   DATA[2646,2] := 2.0;
   DATA[2646,3] := 2.0;
   DATA[2646,4] := 262.3366;
   DATA[2646,5] := 8.393873;
   DATA[2646,6] := 329.2745;
   DATA[2646,7] := 2.455131;
   DATA[2646,8] := 2.0;
   DATA[2646,9] := 2.0;
   DATA[2646,10] := 2.0;
   DATA[2646,11] := 19.69396;
   DATA[2646,12] := 2.209397;
   DATA[2646,13] := 833.5603;
   DATA[2646,14] := 1.0;
   DATA[2646,15] := 2.0;
   DATA[2646,16] := 1.0;
   DATA[2646,17] := 1.0;
   DATA[2646,18] := 1.0;
   DATA[2646,19] := 2.0;
   DATA[2646,20] := 148.808;
   DATA[2646,21] := 155.191;
   DATA[2646,22] := 1.717105;
   DATA[2646,23] := 880.3127;
   DATA[2646,24] := 2.0;
   DATA[2646,25] := 2.0;
   DATA[2646,26] := 7.873815;
   DATA[2646,27] := 144.7578;
   DATA[2646,28] := 261.3753;
   DATA[2646,29] := 12.07383;
   DATA[2646,30] := 1.725711;
   DATA[2646,31] := 1.28705;
   DATA[2646,32] := 0.7352687;
   DATA[2646,33] := 0.3066329;
   DATA[2646,34] := 2.0;
   DATA[2646,35] := 250.2403;
   DATA[2646,36] := 1.665972;
   DATA[2646,37] := 189.022;
   DATA[2646,38] := 0.000128152;
   DATA[2646,39] := 1.0;
   DATA[2646,40] := 1.0;
   DATA[2647,0] := 2.595202;
   DATA[2647,1] := 869.8411;
   DATA[2647,2] := 2.0;
   DATA[2647,3] := 2.0;
   DATA[2647,4] := 262.3366;
   DATA[2647,5] := 8.393873;
   DATA[2647,6] := 329.2745;
   DATA[2647,7] := 2.454362;
   DATA[2647,8] := 2.0;
   DATA[2647,9] := 2.0;
   DATA[2647,10] := 2.0;
   DATA[2647,11] := 19.69396;
   DATA[2647,12] := 2.209397;
   DATA[2647,13] := 833.4402;
   DATA[2647,14] := 1.0;
   DATA[2647,15] := 2.0;
   DATA[2647,16] := 1.0;
   DATA[2647,17] := 1.0;
   DATA[2647,18] := 1.0;
   DATA[2647,19] := 2.0;
   DATA[2647,20] := 148.808;
   DATA[2647,21] := 155.191;
   DATA[2647,22] := 1.718002;
   DATA[2647,23] := 880.8895;
   DATA[2647,24] := 2.0;
   DATA[2647,25] := 2.0;
   DATA[2647,26] := 7.873815;
   DATA[2647,27] := 144.7578;
   DATA[2647,28] := 261.3753;
   DATA[2647,29] := 12.03538;
   DATA[2647,30] := 1.726096;
   DATA[2647,31] := 1.281286;
   DATA[2647,32] := 0.7352687;
   DATA[2647,33] := 0.3065048;
   DATA[2647,34] := 2.0;
   DATA[2647,35] := 250.2403;
   DATA[2647,36] := 1.730048;
   DATA[2647,37] := 189.1182;
   DATA[2647,38] := 0.000128152;
   DATA[2647,39] := 1.0;
   DATA[2647,40] := 1.0;
   DATA[2648,0] := 2.620504;
   DATA[2648,1] := 869.4094;
   DATA[2648,2] := 2.0;
   DATA[2648,3] := 2.0;
   DATA[2648,4] := 262.3366;
   DATA[2648,5] := 8.393873;
   DATA[2648,6] := 329.2745;
   DATA[2648,7] := 2.45308;
   DATA[2648,8] := 2.0;
   DATA[2648,9] := 2.0;
   DATA[2648,10] := 2.0;
   DATA[2648,11] := 19.66835;
   DATA[2648,12] := 2.209397;
   DATA[2648,13] := 833.6404;
   DATA[2648,14] := 1.0;
   DATA[2648,15] := 2.0;
   DATA[2648,16] := 1.0;
   DATA[2648,17] := 1.0;
   DATA[2648,18] := 1.0;
   DATA[2648,19] := 2.0;
   DATA[2648,20] := 148.808;
   DATA[2648,21] := 155.191;
   DATA[2648,22] := 1.718387;
   DATA[2648,23] := 880.8895;
   DATA[2648,24] := 2.0;
   DATA[2648,25] := 2.0;
   DATA[2648,26] := 7.873815;
   DATA[2648,27] := 144.7578;
   DATA[2648,28] := 261.183;
   DATA[2648,29] := 12.03538;
   DATA[2648,30] := 1.726993;
   DATA[2648,31] := 1.28103;
   DATA[2648,32] := 0.7352687;
   DATA[2648,33] := 0.3065048;
   DATA[2648,34] := 2.0;
   DATA[2648,35] := 250.2403;
   DATA[2648,36] := 1.730048;
   DATA[2648,37] := 189.1182;
   DATA[2648,38] := 0.000128152;
   DATA[2648,39] := 1.0;
   DATA[2648,40] := 1.0;
   DATA[2649,0] := 2.656055;
   DATA[2649,1] := 869.4879;
   DATA[2649,2] := 2.0;
   DATA[2649,3] := 2.0;
   DATA[2649,4] := 262.3366;
   DATA[2649,5] := 8.393873;
   DATA[2649,6] := 329.2745;
   DATA[2649,7] := 2.45308;
   DATA[2649,8] := 2.0;
   DATA[2649,9] := 2.0;
   DATA[2649,10] := 2.0;
   DATA[2649,11] := 19.66835;
   DATA[2649,12] := 2.209397;
   DATA[2649,13] := 833.36;
   DATA[2649,14] := 1.0;
   DATA[2649,15] := 2.0;
   DATA[2649,16] := 1.0;
   DATA[2649,17] := 1.0;
   DATA[2649,18] := 1.0;
   DATA[2649,19] := 2.0;
   DATA[2649,20] := 148.808;
   DATA[2649,21] := 155.191;
   DATA[2649,22] := 1.720437;
   DATA[2649,23] := 881.1587;
   DATA[2649,24] := 2.0;
   DATA[2649,25] := 2.0;
   DATA[2649,26] := 7.874776;
   DATA[2649,27] := 144.7578;
   DATA[2649,28] := 261.183;
   DATA[2649,29] := 12.03538;
   DATA[2649,30] := 1.726993;
   DATA[2649,31] := 1.28103;
   DATA[2649,32] := 0.7352687;
   DATA[2649,33] := 0.3065048;
   DATA[2649,34] := 2.0;
   DATA[2649,35] := 250.2403;
   DATA[2649,36] := 1.730048;
   DATA[2649,37] := 189.1182;
   DATA[2649,38] := 0.000128152;
   DATA[2649,39] := 1.0;
   DATA[2649,40] := 1.0;
   DATA[2650,0] := 2.665663;
   DATA[2650,1] := 869.4094;
   DATA[2650,2] := 2.0;
   DATA[2650,3] := 2.0;
   DATA[2650,4] := 262.3366;
   DATA[2650,5] := 8.396757;
   DATA[2650,6] := 329.2745;
   DATA[2650,7] := 2.45308;
   DATA[2650,8] := 2.0;
   DATA[2650,9] := 2.0;
   DATA[2650,10] := 2.0;
   DATA[2650,11] := 19.74198;
   DATA[2650,12] := 2.209397;
   DATA[2650,13] := 833.36;
   DATA[2650,14] := 1.0;
   DATA[2650,15] := 2.0;
   DATA[2650,16] := 1.0;
   DATA[2650,17] := 1.0;
   DATA[2650,18] := 1.0;
   DATA[2650,19] := 2.0;
   DATA[2650,20] := 148.808;
   DATA[2650,21] := 155.191;
   DATA[2650,22] := 1.720437;
   DATA[2650,23] := 881.0433;
   DATA[2650,24] := 2.0;
   DATA[2650,25] := 2.0;
   DATA[2650,26] := 7.874776;
   DATA[2650,27] := 144.7578;
   DATA[2650,28] := 261.183;
   DATA[2650,29] := 12.03538;
   DATA[2650,30] := 1.727634;
   DATA[2650,31] := 1.273601;
   DATA[2650,32] := 0.7352687;
   DATA[2650,33] := 0.3065048;
   DATA[2650,34] := 2.0;
   DATA[2650,35] := 250.3525;
   DATA[2650,36] := 1.730048;
   DATA[2650,37] := 189.1182;
   DATA[2650,38] := 0.000128152;
   DATA[2650,39] := 1.0;
   DATA[2650,40] := 1.0;
   DATA[2651,0] := 2.665663;
   DATA[2651,1] := 869.5271;
   DATA[2651,2] := 2.0;
   DATA[2651,3] := 2.0;
   DATA[2651,4] := 262.3366;
   DATA[2651,5] := 8.396757;
   DATA[2651,6] := 329.1464;
   DATA[2651,7] := 2.454618;
   DATA[2651,8] := 2.0;
   DATA[2651,9] := 2.0;
   DATA[2651,10] := 2.0;
   DATA[2651,11] := 19.74198;
   DATA[2651,12] := 2.209397;
   DATA[2651,13] := 833.5603;
   DATA[2651,14] := 1.0;
   DATA[2651,15] := 2.0;
   DATA[2651,16] := 1.0;
   DATA[2651,17] := 1.0;
   DATA[2651,18] := 1.0;
   DATA[2651,19] := 2.0;
   DATA[2651,20] := 148.808;
   DATA[2651,21] := 155.191;
   DATA[2651,22] := 1.720437;
   DATA[2651,23] := 881.0433;
   DATA[2651,24] := 2.0;
   DATA[2651,25] := 2.0;
   DATA[2651,26] := 7.874776;
   DATA[2651,27] := 144.7578;
   DATA[2651,28] := 261.183;
   DATA[2651,29] := 12.03538;
   DATA[2651,30] := 1.728916;
   DATA[2651,31] := 1.277699;
   DATA[2651,32] := 0.7352687;
   DATA[2651,33] := 0.3065048;
   DATA[2651,34] := 2.0;
   DATA[2651,35] := 250.3525;
   DATA[2651,36] := 1.730048;
   DATA[2651,37] := 189.1182;
   DATA[2651,38] := 0.000128152;
   DATA[2651,39] := 1.0;
   DATA[2651,40] := 1.0;
   DATA[2652,0] := 2.65061;
   DATA[2652,1] := 869.8019;
   DATA[2652,2] := 2.0;
   DATA[2652,3] := 2.0;
   DATA[2652,4] := 262.3366;
   DATA[2652,5] := 8.396757;
   DATA[2652,6] := 329.1464;
   DATA[2652,7] := 2.454618;
   DATA[2652,8] := 2.0;
   DATA[2652,9] := 2.0;
   DATA[2652,10] := 2.0;
   DATA[2652,11] := 19.74198;
   DATA[2652,12] := 2.209397;
   DATA[2652,13] := 833.6004;
   DATA[2652,14] := 1.0;
   DATA[2652,15] := 2.0;
   DATA[2652,16] := 1.0;
   DATA[2652,17] := 1.0;
   DATA[2652,18] := 1.0;
   DATA[2652,19] := 2.0;
   DATA[2652,20] := 148.808;
   DATA[2652,21] := 155.191;
   DATA[2652,22] := 1.720437;
   DATA[2652,23] := 881.1202;
   DATA[2652,24] := 2.0;
   DATA[2652,25] := 2.0;
   DATA[2652,26] := 7.874776;
   DATA[2652,27] := 144.6039;
   DATA[2652,28] := 261.2151;
   DATA[2652,29] := 12.03538;
   DATA[2652,30] := 1.7293;
   DATA[2652,31] := 1.293711;
   DATA[2652,32] := 0.7352687;
   DATA[2652,33] := 0.3065048;
   DATA[2652,34] := 2.0;
   DATA[2652,35] := 250.3525;
   DATA[2652,36] := 1.730048;
   DATA[2652,37] := 189.1182;
   DATA[2652,38] := 0.000128152;
   DATA[2652,39] := 1.0;
   DATA[2652,40] := 1.0;
   DATA[2653,0] := 2.62755;
   DATA[2653,1] := 869.8019;
   DATA[2653,2] := 2.0;
   DATA[2653,3] := 2.0;
   DATA[2653,4] := 262.3366;
   DATA[2653,5] := 8.396757;
   DATA[2653,6] := 329.1464;
   DATA[2653,7] := 2.455515;
   DATA[2653,8] := 2.0;
   DATA[2653,9] := 2.0;
   DATA[2653,10] := 2.0;
   DATA[2653,11] := 19.67476;
   DATA[2653,12] := 2.209397;
   DATA[2653,13] := 833.4802;
   DATA[2653,14] := 1.0;
   DATA[2653,15] := 2.0;
   DATA[2653,16] := 1.0;
   DATA[2653,17] := 1.0;
   DATA[2653,18] := 1.0;
   DATA[2653,19] := 2.0;
   DATA[2653,20] := 148.808;
   DATA[2653,21] := 155.191;
   DATA[2653,22] := 1.720437;
   DATA[2653,23] := 880.8895;
   DATA[2653,24] := 2.0;
   DATA[2653,25] := 2.0;
   DATA[2653,26] := 7.874776;
   DATA[2653,27] := 144.6039;
   DATA[2653,28] := 261.3432;
   DATA[2653,29] := 12.03538;
   DATA[2653,30] := 1.7293;
   DATA[2653,31] := 1.297041;
   DATA[2653,32] := 0.7352687;
   DATA[2653,33] := 0.3065048;
   DATA[2653,34] := 2.0;
   DATA[2653,35] := 250.3525;
   DATA[2653,36] := 1.730048;
   DATA[2653,37] := 189.1182;
   DATA[2653,38] := 0.000128152;
   DATA[2653,39] := 1.0;
   DATA[2653,40] := 1.0;
   DATA[2654,0] := 2.622746;
   DATA[2654,1] := 869.8411;
   DATA[2654,2] := 2.0;
   DATA[2654,3] := 2.0;
   DATA[2654,4] := 262.3366;
   DATA[2654,5] := 8.396757;
   DATA[2654,6] := 329.1464;
   DATA[2654,7] := 2.455515;
   DATA[2654,8] := 2.0;
   DATA[2654,9] := 2.0;
   DATA[2654,10] := 2.0;
   DATA[2654,11] := 19.67476;
   DATA[2654,12] := 2.209397;
   DATA[2654,13] := 833.7606;
   DATA[2654,14] := 1.0;
   DATA[2654,15] := 2.0;
   DATA[2654,16] := 1.0;
   DATA[2654,17] := 1.0;
   DATA[2654,18] := 1.0;
   DATA[2654,19] := 2.0;
   DATA[2654,20] := 148.808;
   DATA[2654,21] := 155.191;
   DATA[2654,22] := 1.720437;
   DATA[2654,23] := 880.7357;
   DATA[2654,24] := 2.0;
   DATA[2654,25] := 2.0;
   DATA[2654,26] := 7.874776;
   DATA[2654,27] := 144.6039;
   DATA[2654,28] := 261.3432;
   DATA[2654,29] := 12.03538;
   DATA[2654,30] := 1.7293;
   DATA[2654,31] := 1.296401;
   DATA[2654,32] := 0.7352687;
   DATA[2654,33] := 0.3065689;
   DATA[2654,34] := 2.0;
   DATA[2654,35] := 250.3525;
   DATA[2654,36] := 1.730048;
   DATA[2654,37] := 189.1342;
   DATA[2654,38] := 0.000128152;
   DATA[2654,39] := 1.0;
   DATA[2654,40] := 1.0;
   DATA[2655,0] := 2.607693;
   DATA[2655,1] := 869.4094;
   DATA[2655,2] := 2.0;
   DATA[2655,3] := 2.0;
   DATA[2655,4] := 262.3366;
   DATA[2655,5] := 8.396757;
   DATA[2655,6] := 329.1464;
   DATA[2655,7] := 2.455515;
   DATA[2655,8] := 2.0;
   DATA[2655,9] := 2.0;
   DATA[2655,10] := 2.0;
   DATA[2655,11] := 19.62033;
   DATA[2655,12] := 2.209397;
   DATA[2655,13] := 833.6404;
   DATA[2655,14] := 1.0;
   DATA[2655,15] := 2.0;
   DATA[2655,16] := 1.0;
   DATA[2655,17] := 1.0;
   DATA[2655,18] := 1.0;
   DATA[2655,19] := 2.0;
   DATA[2655,20] := 148.808;
   DATA[2655,21] := 155.3961;
   DATA[2655,22] := 1.720437;
   DATA[2655,23] := 880.928;
   DATA[2655,24] := 2.0;
   DATA[2655,25] := 2.0;
   DATA[2655,26] := 7.874776;
   DATA[2655,27] := 144.6039;
   DATA[2655,28] := 261.3432;
   DATA[2655,29] := 12.03538;
   DATA[2655,30] := 1.7293;
   DATA[2655,31] := 1.296016;
   DATA[2655,32] := 0.7352687;
   DATA[2655,33] := 0.3066329;
   DATA[2655,34] := 2.0;
   DATA[2655,35] := 250.3525;
   DATA[2655,36] := 1.730048;
   DATA[2655,37] := 189.1662;
   DATA[2655,38] := 0.000128152;
   DATA[2655,39] := 1.0;
   DATA[2655,40] := 1.0;
   DATA[2656,0] := 2.587516;
   DATA[2656,1] := 869.8411;
   DATA[2656,2] := 2.0;
   DATA[2656,3] := 2.0;
   DATA[2656,4] := 262.3366;
   DATA[2656,5] := 8.396757;
   DATA[2656,6] := 329.1464;
   DATA[2656,7] := 2.455515;
   DATA[2656,8] := 2.0;
   DATA[2656,9] := 2.0;
   DATA[2656,10] := 2.0;
   DATA[2656,11] := 19.62033;
   DATA[2656,12] := 2.208884;
   DATA[2656,13] := 833.5603;
   DATA[2656,14] := 1.0;
   DATA[2656,15] := 2.0;
   DATA[2656,16] := 1.0;
   DATA[2656,17] := 1.0;
   DATA[2656,18] := 1.0;
   DATA[2656,19] := 2.0;
   DATA[2656,20] := 148.808;
   DATA[2656,21] := 155.3961;
   DATA[2656,22] := 1.720437;
   DATA[2656,23] := 880.7357;
   DATA[2656,24] := 2.0;
   DATA[2656,25] := 2.0;
   DATA[2656,26] := 7.874776;
   DATA[2656,27] := 144.6039;
   DATA[2656,28] := 261.3432;
   DATA[2656,29] := 12.03538;
   DATA[2656,30] := 1.7293;
   DATA[2656,31] := 1.292558;
   DATA[2656,32] := 0.7352687;
   DATA[2656,33] := 0.3066329;
   DATA[2656,34] := 2.0;
   DATA[2656,35] := 250.3525;
   DATA[2656,36] := 1.730048;
   DATA[2656,37] := 189.1662;
   DATA[2656,38] := 0.000128152;
   DATA[2656,39] := 1.0;
   DATA[2656,40] := 1.0;
   DATA[2657,0] := 2.562854;
   DATA[2657,1] := 870.0767;
   DATA[2657,2] := 2.0;
   DATA[2657,3] := 2.0;
   DATA[2657,4] := 262.3366;
   DATA[2657,5] := 8.396757;
   DATA[2657,6] := 329.1464;
   DATA[2657,7] := 2.455515;
   DATA[2657,8] := 2.0;
   DATA[2657,9] := 2.0;
   DATA[2657,10] := 2.0;
   DATA[2657,11] := 19.57232;
   DATA[2657,12] := 2.208884;
   DATA[2657,13] := 834.0009;
   DATA[2657,14] := 1.0;
   DATA[2657,15] := 2.0;
   DATA[2657,16] := 1.0;
   DATA[2657,17] := 1.0;
   DATA[2657,18] := 1.0;
   DATA[2657,19] := 2.0;
   DATA[2657,20] := 148.808;
   DATA[2657,21] := 155.3961;
   DATA[2657,22] := 1.720437;
   DATA[2657,23] := 880.4666;
   DATA[2657,24] := 2.0;
   DATA[2657,25] := 2.0;
   DATA[2657,26] := 7.873815;
   DATA[2657,27] := 144.6039;
   DATA[2657,28] := 261.3432;
   DATA[2657,29] := 12.03538;
   DATA[2657,30] := 1.7293;
   DATA[2657,31] := 1.291533;
   DATA[2657,32] := 0.7352687;
   DATA[2657,33] := 0.3066329;
   DATA[2657,34] := 2.0;
   DATA[2657,35] := 250.1762;
   DATA[2657,36] := 1.730048;
   DATA[2657,37] := 189.1662;
   DATA[2657,38] := 0.000128152;
   DATA[2657,39] := 1.0;
   DATA[2657,40] := 1.0;
   DATA[2658,0] := 2.537873;
   DATA[2658,1] := 869.7234;
   DATA[2658,2] := 2.0;
   DATA[2658,3] := 2.0;
   DATA[2658,4] := 262.3366;
   DATA[2658,5] := 8.396757;
   DATA[2658,6] := 329.1464;
   DATA[2658,7] := 2.452952;
   DATA[2658,8] := 2.0;
   DATA[2658,9] := 2.0;
   DATA[2658,10] := 2.0;
   DATA[2658,11] := 19.57232;
   DATA[2658,12] := 2.208884;
   DATA[2658,13] := 834.0009;
   DATA[2658,14] := 1.0;
   DATA[2658,15] := 2.0;
   DATA[2658,16] := 1.0;
   DATA[2658,17] := 1.0;
   DATA[2658,18] := 1.0;
   DATA[2658,19] := 2.0;
   DATA[2658,20] := 148.808;
   DATA[2658,21] := 155.3961;
   DATA[2658,22] := 1.720437;
   DATA[2658,23] := 880.8511;
   DATA[2658,24] := 2.0;
   DATA[2658,25] := 2.0;
   DATA[2658,26] := 7.873815;
   DATA[2658,27] := 144.6039;
   DATA[2658,28] := 261.3432;
   DATA[2658,29] := 12.03538;
   DATA[2658,30] := 1.7293;
   DATA[2658,31] := 1.291533;
   DATA[2658,32] := 0.7352687;
   DATA[2658,33] := 0.3066329;
   DATA[2658,34] := 2.0;
   DATA[2658,35] := 250.1762;
   DATA[2658,36] := 1.730048;
   DATA[2658,37] := 188.9419;
   DATA[2658,38] := 0.000128152;
   DATA[2658,39] := 1.0;
   DATA[2658,40] := 1.0;
   DATA[2659,0] := 2.521218;
   DATA[2659,1] := 869.8019;
   DATA[2659,2] := 2.0;
   DATA[2659,3] := 2.0;
   DATA[2659,4] := 262.3366;
   DATA[2659,5] := 8.396757;
   DATA[2659,6] := 329.1464;
   DATA[2659,7] := 2.452952;
   DATA[2659,8] := 2.0;
   DATA[2659,9] := 2.0;
   DATA[2659,10] := 2.0;
   DATA[2659,11] := 19.62674;
   DATA[2659,12] := 2.209653;
   DATA[2659,13] := 834.0009;
   DATA[2659,14] := 1.0;
   DATA[2659,15] := 2.0;
   DATA[2659,16] := 1.0;
   DATA[2659,17] := 1.0;
   DATA[2659,18] := 1.0;
   DATA[2659,19] := 2.0;
   DATA[2659,20] := 148.808;
   DATA[2659,21] := 155.3961;
   DATA[2659,22] := 1.718002;
   DATA[2659,23] := 880.6588;
   DATA[2659,24] := 2.0;
   DATA[2659,25] := 2.0;
   DATA[2659,26] := 7.872853;
   DATA[2659,27] := 144.6039;
   DATA[2659,28] := 261.3432;
   DATA[2659,29] := 12.03538;
   DATA[2659,30] := 1.7293;
   DATA[2659,31] := 1.291533;
   DATA[2659,32] := 0.7352687;
   DATA[2659,33] := 0.3066329;
   DATA[2659,34] := 2.0;
   DATA[2659,35] := 249.9519;
   DATA[2659,36] := 1.730048;
   DATA[2659,37] := 188.8618;
   DATA[2659,38] := 0.000128152;
   DATA[2659,39] := 1.0;
   DATA[2659,40] := 1.0;
   DATA[2660,0] := 2.500721;
   DATA[2660,1] := 869.9196;
   DATA[2660,2] := 2.0;
   DATA[2660,3] := 2.0;
   DATA[2660,4] := 262.3366;
   DATA[2660,5] := 8.396757;
   DATA[2660,6] := 329.1464;
   DATA[2660,7] := 2.452952;
   DATA[2660,8] := 2.0;
   DATA[2660,9] := 2.0;
   DATA[2660,10] := 2.0;
   DATA[2660,11] := 19.62674;
   DATA[2660,12] := 2.209653;
   DATA[2660,13] := 834.1611;
   DATA[2660,14] := 1.0;
   DATA[2660,15] := 2.0;
   DATA[2660,16] := 1.0;
   DATA[2660,17] := 1.0;
   DATA[2660,18] := 1.0;
   DATA[2660,19] := 2.0;
   DATA[2660,20] := 148.808;
   DATA[2660,21] := 155.3961;
   DATA[2660,22] := 1.717361;
   DATA[2660,23] := 881.0818;
   DATA[2660,24] := 2.0;
   DATA[2660,25] := 2.0;
   DATA[2660,26] := 7.872853;
   DATA[2660,27] := 144.6039;
   DATA[2660,28] := 261.3432;
   DATA[2660,29] := 12.03538;
   DATA[2660,30] := 1.7293;
   DATA[2660,31] := 1.28436;
   DATA[2660,32] := 0.7352687;
   DATA[2660,33] := 0.3066329;
   DATA[2660,34] := 2.0;
   DATA[2660,35] := 249.9519;
   DATA[2660,36] := 1.730048;
   DATA[2660,37] := 188.8618;
   DATA[2660,38] := 0.000128152;
   DATA[2660,39] := 1.0;
   DATA[2660,40] := 1.0;
   DATA[2661,0] := 2.483426;
   DATA[2661,1] := 870.1159;
   DATA[2661,2] := 2.0;
   DATA[2661,3] := 2.0;
   DATA[2661,4] := 262.3366;
   DATA[2661,5] := 8.396757;
   DATA[2661,6] := 329.1464;
   DATA[2661,7] := 2.452952;
   DATA[2661,8] := 2.0;
   DATA[2661,9] := 2.0;
   DATA[2661,10] := 2.0;
   DATA[2661,11] := 19.62674;
   DATA[2661,12] := 2.209653;
   DATA[2661,13] := 833.6004;
   DATA[2661,14] := 1.0;
   DATA[2661,15] := 2.0;
   DATA[2661,16] := 1.0;
   DATA[2661,17] := 1.0;
   DATA[2661,18] := 1.0;
   DATA[2661,19] := 2.0;
   DATA[2661,20] := 148.808;
   DATA[2661,21] := 155.3961;
   DATA[2661,22] := 1.717233;
   DATA[2661,23] := 880.7742;
   DATA[2661,24] := 2.0;
   DATA[2661,25] := 2.0;
   DATA[2661,26] := 7.872853;
   DATA[2661,27] := 144.7065;
   DATA[2661,28] := 261.3432;
   DATA[2661,29] := 12.03538;
   DATA[2661,30] := 1.7293;
   DATA[2661,31] := 1.286922;
   DATA[2661,32] := 0.7352687;
   DATA[2661,33] := 0.3066329;
   DATA[2661,34] := 2.0;
   DATA[2661,35] := 249.9519;
   DATA[2661,36] := 1.730048;
   DATA[2661,37] := 188.8618;
   DATA[2661,38] := 0.000128152;
   DATA[2661,39] := 1.0;
   DATA[2661,40] := 1.0;
   DATA[2662,0] := 2.468052;
   DATA[2662,1] := 870.2729;
   DATA[2662,2] := 2.0;
   DATA[2662,3] := 2.0;
   DATA[2662,4] := 262.3366;
   DATA[2662,5] := 8.396757;
   DATA[2662,6] := 329.1464;
   DATA[2662,7] := 2.452952;
   DATA[2662,8] := 2.0;
   DATA[2662,9] := 2.0;
   DATA[2662,10] := 2.0;
   DATA[2662,11] := 19.67476;
   DATA[2662,12] := 2.208756;
   DATA[2662,13] := 833.5603;
   DATA[2662,14] := 1.0;
   DATA[2662,15] := 2.0;
   DATA[2662,16] := 1.0;
   DATA[2662,17] := 1.0;
   DATA[2662,18] := 1.0;
   DATA[2662,19] := 2.0;
   DATA[2662,20] := 148.808;
   DATA[2662,21] := 155.3961;
   DATA[2662,22] := 1.717233;
   DATA[2662,23] := 880.5819;
   DATA[2662,24] := 2.0;
   DATA[2662,25] := 2.0;
   DATA[2662,26] := 7.872853;
   DATA[2662,27] := 144.7065;
   DATA[2662,28] := 261.3432;
   DATA[2662,29] := 12.03538;
   DATA[2662,30] := 1.7293;
   DATA[2662,31] := 1.301012;
   DATA[2662,32] := 0.7352687;
   DATA[2662,33] := 0.3066329;
   DATA[2662,34] := 2.0;
   DATA[2662,35] := 249.9519;
   DATA[2662,36] := 1.730048;
   DATA[2662,37] := 188.8618;
   DATA[2662,38] := 0.000128152;
   DATA[2662,39] := 1.0;
   DATA[2662,40] := 1.0;
   DATA[2663,0] := 2.449156;
   DATA[2663,1] := 870.5084;
   DATA[2663,2] := 2.0;
   DATA[2663,3] := 2.0;
   DATA[2663,4] := 262.3366;
   DATA[2663,5] := 8.396757;
   DATA[2663,6] := 329.1464;
   DATA[2663,7] := 2.452952;
   DATA[2663,8] := 2.0;
   DATA[2663,9] := 2.0;
   DATA[2663,10] := 2.0;
   DATA[2663,11] := 19.69396;
   DATA[2663,12] := 2.208756;
   DATA[2663,13] := 833.8007;
   DATA[2663,14] := 1.0;
   DATA[2663,15] := 2.0;
   DATA[2663,16] := 1.0;
   DATA[2663,17] := 1.0;
   DATA[2663,18] := 1.0;
   DATA[2663,19] := 2.0;
   DATA[2663,20] := 148.808;
   DATA[2663,21] := 155.3961;
   DATA[2663,22] := 1.717233;
   DATA[2663,23] := 880.6973;
   DATA[2663,24] := 2.0;
   DATA[2663,25] := 2.0;
   DATA[2663,26] := 7.872853;
   DATA[2663,27] := 144.7065;
   DATA[2663,28] := 261.3432;
   DATA[2663,29] := 12.03538;
   DATA[2663,30] := 1.7293;
   DATA[2663,31] := 1.296529;
   DATA[2663,32] := 0.7352687;
   DATA[2663,33] := 0.3066329;
   DATA[2663,34] := 2.0;
   DATA[2663,35] := 249.9519;
   DATA[2663,36] := 1.730048;
   DATA[2663,37] := 188.8618;
   DATA[2663,38] := 0.000128152;
   DATA[2663,39] := 1.0;
   DATA[2663,40] := 1.0;
   DATA[2664,0] := 2.436665;
   DATA[2664,1] := 870.4299;
   DATA[2664,2] := 2.0;
   DATA[2664,3] := 2.0;
   DATA[2664,4] := 262.3366;
   DATA[2664,5] := 8.396757;
   DATA[2664,6] := 329.1464;
   DATA[2664,7] := 2.452055;
   DATA[2664,8] := 2.0;
   DATA[2664,9] := 2.0;
   DATA[2664,10] := 2.0;
   DATA[2664,11] := 19.69396;
   DATA[2664,12] := 2.206322;
   DATA[2664,13] := 834.0009;
   DATA[2664,14] := 1.0;
   DATA[2664,15] := 2.0;
   DATA[2664,16] := 1.0;
   DATA[2664,17] := 1.0;
   DATA[2664,18] := 1.0;
   DATA[2664,19] := 2.0;
   DATA[2664,20] := 148.808;
   DATA[2664,21] := 155.3961;
   DATA[2664,22] := 1.717233;
   DATA[2664,23] := 880.7357;
   DATA[2664,24] := 2.0;
   DATA[2664,25] := 2.0;
   DATA[2664,26] := 7.872853;
   DATA[2664,27] := 144.7065;
   DATA[2664,28] := 261.3432;
   DATA[2664,29] := 12.03538;
   DATA[2664,30] := 1.726352;
   DATA[2664,31] := 1.3005;
   DATA[2664,32] := 0.7352687;
   DATA[2664,33] := 0.3066329;
   DATA[2664,34] := 2.0;
   DATA[2664,35] := 250.016;
   DATA[2664,36] := 1.730048;
   DATA[2664,37] := 188.8618;
   DATA[2664,38] := 0.000128152;
   DATA[2664,39] := 1.0;
   DATA[2664,40] := 1.0;
   DATA[2665,0] := 2.431861;
   DATA[2665,1] := 870.5869;
   DATA[2665,2] := 2.0;
   DATA[2665,3] := 2.0;
   DATA[2665,4] := 262.3366;
   DATA[2665,5] := 8.396757;
   DATA[2665,6] := 329.1464;
   DATA[2665,7] := 2.451799;
   DATA[2665,8] := 2.0;
   DATA[2665,9] := 2.0;
   DATA[2665,10] := 2.0;
   DATA[2665,11] := 19.69396;
   DATA[2665,12] := 2.206322;
   DATA[2665,13] := 834.4415;
   DATA[2665,14] := 1.0;
   DATA[2665,15] := 2.0;
   DATA[2665,16] := 1.0;
   DATA[2665,17] := 1.0;
   DATA[2665,18] := 1.0;
   DATA[2665,19] := 2.0;
   DATA[2665,20] := 148.808;
   DATA[2665,21] := 155.3961;
   DATA[2665,22] := 1.717233;
   DATA[2665,23] := 881.2356;
   DATA[2665,24] := 2.0;
   DATA[2665,25] := 2.0;
   DATA[2665,26] := 7.872853;
   DATA[2665,27] := 144.7065;
   DATA[2665,28] := 261.3432;
   DATA[2665,29] := 12.03538;
   DATA[2665,30] := 1.726352;
   DATA[2665,31] := 1.3119;
   DATA[2665,32] := 0.7352687;
   DATA[2665,33] := 0.3066329;
   DATA[2665,34] := 2.0;
   DATA[2665,35] := 250.0961;
   DATA[2665,36] := 1.730048;
   DATA[2665,37] := 188.8618;
   DATA[2665,38] := 0.000128152;
   DATA[2665,39] := 1.0;
   DATA[2665,40] := 1.0;
   DATA[2666,0] := 2.431861;
   DATA[2666,1] := 870.4692;
   DATA[2666,2] := 2.0;
   DATA[2666,3] := 2.0;
   DATA[2666,4] := 262.3366;
   DATA[2666,5] := 8.396757;
   DATA[2666,6] := 329.1464;
   DATA[2666,7] := 2.451799;
   DATA[2666,8] := 2.0;
   DATA[2666,9] := 2.0;
   DATA[2666,10] := 2.0;
   DATA[2666,11] := 19.72598;
   DATA[2666,12] := 2.206322;
   DATA[2666,13] := 834.4415;
   DATA[2666,14] := 1.0;
   DATA[2666,15] := 2.0;
   DATA[2666,16] := 1.0;
   DATA[2666,17] := 1.0;
   DATA[2666,18] := 1.0;
   DATA[2666,19] := 2.0;
   DATA[2666,20] := 148.808;
   DATA[2666,21] := 155.3961;
   DATA[2666,22] := 1.717233;
   DATA[2666,23] := 881.4663;
   DATA[2666,24] := 2.0;
   DATA[2666,25] := 2.0;
   DATA[2666,26] := 7.872853;
   DATA[2666,27] := 144.7065;
   DATA[2666,28] := 261.3432;
   DATA[2666,29] := 12.03538;
   DATA[2666,30] := 1.726352;
   DATA[2666,31] := 1.30652;
   DATA[2666,32] := 0.7352687;
   DATA[2666,33] := 0.3066329;
   DATA[2666,34] := 2.0;
   DATA[2666,35] := 250.0961;
   DATA[2666,36] := 1.730048;
   DATA[2666,37] := 188.8618;
   DATA[2666,38] := 0.000128152;
   DATA[2666,39] := 1.0;
   DATA[2666,40] := 1.0;
   DATA[2667,0] := 2.455882;
   DATA[2667,1] := 870.5869;
   DATA[2667,2] := 2.0;
   DATA[2667,3] := 2.0;
   DATA[2667,4] := 262.3366;
   DATA[2667,5] := 8.396757;
   DATA[2667,6] := 329.1464;
   DATA[2667,7] := 2.455131;
   DATA[2667,8] := 2.0;
   DATA[2667,9] := 2.0;
   DATA[2667,10] := 2.0;
   DATA[2667,11] := 19.74198;
   DATA[2667,12] := 2.20645;
   DATA[2667,13] := 834.802;
   DATA[2667,14] := 1.0;
   DATA[2667,15] := 2.0;
   DATA[2667,16] := 1.0;
   DATA[2667,17] := 1.0;
   DATA[2667,18] := 1.0;
   DATA[2667,19] := 2.0;
   DATA[2667,20] := 148.808;
   DATA[2667,21] := 155.3961;
   DATA[2667,22] := 1.719156;
   DATA[2667,23] := 882.0431;
   DATA[2667,24] := 2.0;
   DATA[2667,25] := 2.0;
   DATA[2667,26] := 7.872853;
   DATA[2667,27] := 144.7065;
   DATA[2667,28] := 261.3432;
   DATA[2667,29] := 12.03538;
   DATA[2667,30] := 1.726352;
   DATA[2667,31] := 1.311387;
   DATA[2667,32] := 0.7352687;
   DATA[2667,33] := 0.3066329;
   DATA[2667,34] := 2.0;
   DATA[2667,35] := 250.1442;
   DATA[2667,36] := 1.730048;
   DATA[2667,37] := 188.8618;
   DATA[2667,38] := 0.000128152;
   DATA[2667,39] := 1.0;
   DATA[2667,40] := 1.0;
   DATA[2668,0] := 2.50008;
   DATA[2668,1] := 870.3907;
   DATA[2668,2] := 2.0;
   DATA[2668,3] := 2.0;
   DATA[2668,4] := 262.3366;
   DATA[2668,5] := 8.396757;
   DATA[2668,6] := 329.1464;
   DATA[2668,7] := 2.455131;
   DATA[2668,8] := 2.0;
   DATA[2668,9] := 2.0;
   DATA[2668,10] := 2.0;
   DATA[2668,11] := 19.75799;
   DATA[2668,12] := 2.209909;
   DATA[2668,13] := 834.802;
   DATA[2668,14] := 1.0;
   DATA[2668,15] := 2.0;
   DATA[2668,16] := 1.0;
   DATA[2668,17] := 1.0;
   DATA[2668,18] := 1.0;
   DATA[2668,19] := 2.0;
   DATA[2668,20] := 148.808;
   DATA[2668,21] := 155.3961;
   DATA[2668,22] := 1.719156;
   DATA[2668,23] := 882.1969;
   DATA[2668,24] := 2.0;
   DATA[2668,25] := 2.0;
   DATA[2668,26] := 7.872853;
   DATA[2668,27] := 144.7065;
   DATA[2668,28] := 261.3432;
   DATA[2668,29] := 12.03538;
   DATA[2668,30] := 1.726352;
   DATA[2668,31] := 1.313949;
   DATA[2668,32] := 0.7352687;
   DATA[2668,33] := 0.3066329;
   DATA[2668,34] := 2.0;
   DATA[2668,35] := 250.3044;
   DATA[2668,36] := 1.730048;
   DATA[2668,37] := 189.0381;
   DATA[2668,38] := 0.000128152;
   DATA[2668,39] := 1.0;
   DATA[2668,40] := 1.0;
   DATA[2669,0] := 2.537873;
   DATA[2669,1] := 870.7047;
   DATA[2669,2] := 2.0;
   DATA[2669,3] := 2.0;
   DATA[2669,4] := 262.3366;
   DATA[2669,5] := 8.396757;
   DATA[2669,6] := 329.1464;
   DATA[2669,7] := 2.455131;
   DATA[2669,8] := 2.0;
   DATA[2669,9] := 2.0;
   DATA[2669,10] := 2.0;
   DATA[2669,11] := 19.7964;
   DATA[2669,12] := 2.209909;
   DATA[2669,13] := 835.1625;
   DATA[2669,14] := 1.0;
   DATA[2669,15] := 2.0;
   DATA[2669,16] := 1.0;
   DATA[2669,17] := 1.0;
   DATA[2669,18] := 1.0;
   DATA[2669,19] := 2.0;
   DATA[2669,20] := 148.808;
   DATA[2669,21] := 155.3961;
   DATA[2669,22] := 1.719156;
   DATA[2669,23] := 882.2354;
   DATA[2669,24] := 2.0;
   DATA[2669,25] := 2.0;
   DATA[2669,26] := 7.874135;
   DATA[2669,27] := 144.7065;
   DATA[2669,28] := 261.3432;
   DATA[2669,29] := 12.03538;
   DATA[2669,30] := 1.726352;
   DATA[2669,31] := 1.311643;
   DATA[2669,32] := 0.7352687;
   DATA[2669,33] := 0.3066329;
   DATA[2669,34] := 2.0;
   DATA[2669,35] := 250.3044;
   DATA[2669,36] := 1.730048;
   DATA[2669,37] := 189.0541;
   DATA[2669,38] := 0.000128152;
   DATA[2669,39] := 1.0;
   DATA[2669,40] := 1.0;
   DATA[2670,0] := 2.585594;
   DATA[2670,1] := 871.058;
   DATA[2670,2] := 2.0;
   DATA[2670,3] := 2.0;
   DATA[2670,4] := 262.3366;
   DATA[2670,5] := 8.396757;
   DATA[2670,6] := 329.1464;
   DATA[2670,7] := 2.455131;
   DATA[2670,8] := 2.0;
   DATA[2670,9] := 2.0;
   DATA[2670,10] := 2.0;
   DATA[2670,11] := 19.7964;
   DATA[2670,12] := 2.209909;
   DATA[2670,13] := 835.1625;
   DATA[2670,14] := 1.0;
   DATA[2670,15] := 2.0;
   DATA[2670,16] := 1.0;
   DATA[2670,17] := 1.0;
   DATA[2670,18] := 1.0;
   DATA[2670,19] := 2.0;
   DATA[2670,20] := 148.808;
   DATA[2670,21] := 155.3961;
   DATA[2670,22] := 1.717105;
   DATA[2670,23] := 882.3892;
   DATA[2670,24] := 2.0;
   DATA[2670,25] := 2.0;
   DATA[2670,26] := 7.874135;
   DATA[2670,27] := 144.7065;
   DATA[2670,28] := 261.3432;
   DATA[2670,29] := 12.03538;
   DATA[2670,30] := 1.726352;
   DATA[2670,31] := 1.288587;
   DATA[2670,32] := 0.7352687;
   DATA[2670,33] := 0.3066329;
   DATA[2670,34] := 2.0;
   DATA[2670,35] := 250.3044;
   DATA[2670,36] := 1.730048;
   DATA[2670,37] := 189.1182;
   DATA[2670,38] := 0.000128152;
   DATA[2670,39] := 1.0;
   DATA[2670,40] := 1.0;
   DATA[2671,0] := 2.618903;
   DATA[2671,1] := 870.7047;
   DATA[2671,2] := 2.0;
   DATA[2671,3] := 2.0;
   DATA[2671,4] := 262.3366;
   DATA[2671,5] := 8.396757;
   DATA[2671,6] := 329.1464;
   DATA[2671,7] := 2.456156;
   DATA[2671,8] := 2.0;
   DATA[2671,9] := 2.0;
   DATA[2671,10] := 2.0;
   DATA[2671,11] := 19.7804;
   DATA[2671,12] := 2.209909;
   DATA[2671,13] := 835.2025;
   DATA[2671,14] := 1.0;
   DATA[2671,15] := 2.0;
   DATA[2671,16] := 1.0;
   DATA[2671,17] := 1.0;
   DATA[2671,18] := 1.0;
   DATA[2671,19] := 2.0;
   DATA[2671,20] := 148.808;
   DATA[2671,21] := 155.3961;
   DATA[2671,22] := 1.717105;
   DATA[2671,23] := 882.6967;
   DATA[2671,24] := 2.0;
   DATA[2671,25] := 2.0;
   DATA[2671,26] := 7.874135;
   DATA[2671,27] := 144.7065;
   DATA[2671,28] := 261.3432;
   DATA[2671,29] := 12.03538;
   DATA[2671,30] := 1.726352;
   DATA[2671,31] := 1.27296;
   DATA[2671,32] := 0.7352687;
   DATA[2671,33] := 0.3066329;
   DATA[2671,34] := 2.0;
   DATA[2671,35] := 250.3044;
   DATA[2671,36] := 1.730048;
   DATA[2671,37] := 189.1182;
   DATA[2671,38] := 0.000128152;
   DATA[2671,39] := 1.0;
   DATA[2671,40] := 1.0;
   DATA[2672,0] := 2.644845;
   DATA[2672,1] := 871.2542;
   DATA[2672,2] := 2.0;
   DATA[2672,3] := 2.0;
   DATA[2672,4] := 262.3366;
   DATA[2672,5] := 8.396757;
   DATA[2672,6] := 329.1464;
   DATA[2672,7] := 2.456156;
   DATA[2672,8] := 2.0;
   DATA[2672,9] := 2.0;
   DATA[2672,10] := 2.0;
   DATA[2672,11] := 19.73558;
   DATA[2672,12] := 2.209909;
   DATA[2672,13] := 835.2827;
   DATA[2672,14] := 1.0;
   DATA[2672,15] := 2.0;
   DATA[2672,16] := 1.0;
   DATA[2672,17] := 1.0;
   DATA[2672,18] := 1.0;
   DATA[2672,19] := 2.0;
   DATA[2672,20] := 148.808;
   DATA[2672,21] := 155.3961;
   DATA[2672,22] := 1.717105;
   DATA[2672,23] := 882.8121;
   DATA[2672,24] := 2.0;
   DATA[2672,25] := 2.0;
   DATA[2672,26] := 7.874135;
   DATA[2672,27] := 144.7065;
   DATA[2672,28] := 261.3432;
   DATA[2672,29] := 12.03538;
   DATA[2672,30] := 1.726352;
   DATA[2672,31] := 1.265915;
   DATA[2672,32] := 0.7352687;
   DATA[2672,33] := 0.3066329;
   DATA[2672,34] := 2.0;
   DATA[2672,35] := 250.3044;
   DATA[2672,36] := 1.730048;
   DATA[2672,37] := 188.9419;
   DATA[2672,38] := 0.000128152;
   DATA[2672,39] := 1.0;
   DATA[2672,40] := 1.0;
   DATA[2673,0] := 2.658937;
   DATA[2673,1] := 871.058;
   DATA[2673,3] := 2.0;
   DATA[2673,4] := 262.3366;
   DATA[2673,5] := 8.396757;
   DATA[2673,6] := 329.1464;
   DATA[2673,7] := 2.456156;
   DATA[2673,8] := 2.0;
   DATA[2673,9] := 2.0;
   DATA[2673,10] := 2.0;
   DATA[2673,11] := 19.71637;
   DATA[2673,12] := 2.211959;
   DATA[2673,13] := 835.6832;
   DATA[2673,14] := 1.0;
   DATA[2673,15] := 2.0;
   DATA[2673,16] := 1.0;
   DATA[2673,17] := 1.0;
   DATA[2673,18] := 1.0;
   DATA[2673,19] := 2.0;
   DATA[2673,20] := 148.808;
   DATA[2673,21] := 155.3961;
   DATA[2673,22] := 1.717105;
   DATA[2673,23] := 882.6967;
   DATA[2673,24] := 2.0;
   DATA[2673,25] := 2.0;
   DATA[2673,26] := 7.874135;
   DATA[2673,27] := 144.7065;
   DATA[2673,28] := 261.3432;
   DATA[2673,29] := 12.03538;
   DATA[2673,30] := 1.728659;
   DATA[2673,31] := 1.261944;
   DATA[2673,32] := 0.7352687;
   DATA[2673,33] := 0.3066329;
   DATA[2673,34] := 2.0;
   DATA[2673,35] := 250.3044;
   DATA[2673,36] := 1.730048;
   DATA[2673,37] := 188.9419;
   DATA[2673,38] := 0.000128152;
   DATA[2673,39] := 1.0;
   DATA[2673,40] := 1.0;
   DATA[2674,0] := 2.658937;
   DATA[2674,1] := 871.0972;
   DATA[2674,3] := 2.0;
   DATA[2674,4] := 262.3366;
   DATA[2674,5] := 8.396757;
   DATA[2674,6] := 329.1464;
   DATA[2674,7] := 2.453978;
   DATA[2674,8] := 2.0;
   DATA[2674,9] := 2.0;
   DATA[2674,10] := 2.0;
   DATA[2674,11] := 19.71637;
   DATA[2674,12] := 2.212215;
   DATA[2674,13] := 835.563;
   DATA[2674,14] := 1.0;
   DATA[2674,15] := 2.0;
   DATA[2674,16] := 1.0;
   DATA[2674,17] := 1.0;
   DATA[2674,18] := 1.0;
   DATA[2674,19] := 2.0;
   DATA[2674,20] := 148.808;
   DATA[2674,21] := 155.3961;
   DATA[2674,22] := 1.717105;
   DATA[2674,23] := 882.889;
   DATA[2674,24] := 2.0;
   DATA[2674,25] := 2.0;
   DATA[2674,26] := 7.874135;
   DATA[2674,27] := 144.7065;
   DATA[2674,28] := 261.3432;
   DATA[2674,29] := 12.03538;
   DATA[2674,30] := 1.728916;
   DATA[2674,31] := 1.276419;
   DATA[2674,32] := 0.7352687;
   DATA[2674,33] := 0.3066329;
   DATA[2674,34] := 2.0;
   DATA[2674,35] := 250.1442;
   DATA[2674,36] := 1.730048;
   DATA[2674,37] := 188.9419;
   DATA[2674,38] := 0.000128152;
   DATA[2674,39] := 1.0;
   DATA[2674,40] := 1.0;
   DATA[2675,0] := 2.639721;
   DATA[2675,1] := 871.215;
   DATA[2675,3] := 2.0;
   DATA[2675,4] := 262.3366;
   DATA[2675,5] := 8.396757;
   DATA[2675,6] := 329.1464;
   DATA[2675,7] := 2.452952;
   DATA[2675,8] := 2.0;
   DATA[2675,9] := 2.0;
   DATA[2675,10] := 2.0;
   DATA[2675,11] := 19.71637;
   DATA[2675,12] := 2.212215;
   DATA[2675,13] := 835.4028;
   DATA[2675,14] := 1.0;
   DATA[2675,15] := 2.0;
   DATA[2675,16] := 1.0;
   DATA[2675,17] := 1.0;
   DATA[2675,18] := 1.0;
   DATA[2675,19] := 2.0;
   DATA[2675,20] := 148.808;
   DATA[2675,21] := 155.3961;
   DATA[2675,22] := 1.717105;
   DATA[2675,23] := 882.6198;
   DATA[2675,24] := 2.0;
   DATA[2675,25] := 2.0;
   DATA[2675,26] := 7.874135;
   DATA[2675,27] := 144.7065;
   DATA[2675,28] := 261.3432;
   DATA[2675,29] := 11.72776;
   DATA[2675,30] := 1.728916;
   DATA[2675,31] := 1.28167;
   DATA[2675,32] := 0.7352687;
   DATA[2675,33] := 0.3066329;
   DATA[2675,34] := 2.0;
   DATA[2675,35] := 250.1442;
   DATA[2675,36] := 1.730048;
   DATA[2675,37] := 188.9419;
   DATA[2675,38] := 0.000128152;
   DATA[2675,39] := 1.0;
   DATA[2675,40] := 1.0;
   DATA[2676,0] := 2.633635;
   DATA[2676,1] := 870.9794;
   DATA[2676,3] := 2.0;
   DATA[2676,4] := 262.3366;
   DATA[2676,5] := 8.396757;
   DATA[2676,6] := 329.1464;
   DATA[2676,7] := 2.452952;
   DATA[2676,8] := 2.0;
   DATA[2676,9] := 2.0;
   DATA[2676,10] := 2.0;
   DATA[2676,11] := 19.71637;
   DATA[2676,12] := 2.209397;
   DATA[2676,13] := 835.6031;
   DATA[2676,14] := 1.0;
   DATA[2676,15] := 2.0;
   DATA[2676,16] := 1.0;
   DATA[2676,17] := 1.0;
   DATA[2676,18] := 1.0;
   DATA[2676,19] := 2.0;
   DATA[2676,20] := 148.808;
   DATA[2676,21] := 155.5242;
   DATA[2676,22] := 1.717105;
   DATA[2676,23] := 882.5814;
   DATA[2676,24] := 2.0;
   DATA[2676,25] := 2.0;
   DATA[2676,26] := 7.874135;
   DATA[2676,27] := 144.7065;
   DATA[2676,28] := 261.3432;
   DATA[2676,29] := 11.72776;
   DATA[2676,30] := 1.728916;
   DATA[2676,31] := 1.276547;
   DATA[2676,32] := 0.7352687;
   DATA[2676,33] := 0.3066329;
   DATA[2676,34] := 2.0;
   DATA[2676,35] := 250.3525;
   DATA[2676,36] := 1.730048;
   DATA[2676,37] := 189.1182;
   DATA[2676,38] := 0.000128152;
   DATA[2676,39] := 1.0;
   DATA[2676,40] := 1.0;
   DATA[2677,0] := 2.633635;
   DATA[2677,1] := 870.6654;
   DATA[2677,3] := 2.0;
   DATA[2677,4] := 262.3366;
   DATA[2677,5] := 8.396757;
   DATA[2677,6] := 329.1464;
   DATA[2677,7] := 2.452952;
   DATA[2677,8] := 2.0;
   DATA[2677,9] := 2.0;
   DATA[2677,10] := 2.0;
   DATA[2677,11] := 19.71637;
   DATA[2677,12] := 2.209397;
   DATA[2677,13] := 835.4429;
   DATA[2677,14] := 1.0;
   DATA[2677,15] := 2.0;
   DATA[2677,16] := 1.0;
   DATA[2677,17] := 1.0;
   DATA[2677,18] := 1.0;
   DATA[2677,19] := 2.0;
   DATA[2677,20] := 148.808;
   DATA[2677,21] := 155.5242;
   DATA[2677,22] := 1.718515;
   DATA[2677,23] := 882.6967;
   DATA[2677,24] := 2.0;
   DATA[2677,25] := 2.0;
   DATA[2677,26] := 7.874135;
   DATA[2677,27] := 144.7065;
   DATA[2677,28] := 261.3432;
   DATA[2677,29] := 11.72776;
   DATA[2677,30] := 1.730838;
   DATA[2677,31] := 1.280902;
   DATA[2677,32] := 0.7352687;
   DATA[2677,33] := 0.3084905;
   DATA[2677,34] := 2.0;
   DATA[2677,35] := 250.3525;
   DATA[2677,36] := 1.730048;
   DATA[2677,37] := 189.1182;
   DATA[2677,38] := 0.000128152;
   DATA[2677,39] := 1.0;
   DATA[2677,40] := 1.0;
   DATA[2678,0] := 2.625628;
   DATA[2678,1] := 870.6654;
   DATA[2678,3] := 2.0;
   DATA[2678,4] := 262.3366;
   DATA[2678,5] := 8.396757;
   DATA[2678,6] := 329.1464;
   DATA[2678,7] := 2.452952;
   DATA[2678,8] := 2.0;
   DATA[2678,9] := 2.0;
   DATA[2678,10] := 2.0;
   DATA[2678,11] := 19.73878;
   DATA[2678,12] := 2.209397;
   DATA[2678,13] := 835.3627;
   DATA[2678,14] := 1.0;
   DATA[2678,15] := 2.0;
   DATA[2678,16] := 1.0;
   DATA[2678,17] := 1.0;
   DATA[2678,18] := 1.0;
   DATA[2678,19] := 2.0;
   DATA[2678,20] := 148.808;
   DATA[2678,21] := 155.5242;
   DATA[2678,22] := 1.718515;
   DATA[2678,23] := 882.6583;
   DATA[2678,24] := 2.0;
   DATA[2678,25] := 2.0;
   DATA[2678,26] := 7.874135;
   DATA[2678,27] := 144.7065;
   DATA[2678,28] := 261.3432;
   DATA[2678,29] := 12.07383;
   DATA[2678,30] := 1.731735;
   DATA[2678,31] := 1.288203;
   DATA[2678,32] := 0.7352687;
   DATA[2678,33] := 0.3084905;
   DATA[2678,34] := 2.0;
   DATA[2678,35] := 250.4967;
   DATA[2678,36] := 1.730048;
   DATA[2678,37] := 189.2624;
   DATA[2678,38] := 0.000128152;
   DATA[2678,39] := 1.0;
   DATA[2678,40] := 1.0;
   DATA[2679,0] := 2.600006;
   DATA[2679,1] := 871.058;
   DATA[2679,3] := 2.0;
   DATA[2679,4] := 262.3366;
   DATA[2679,5] := 8.396757;
   DATA[2679,6] := 329.1464;
   DATA[2679,7] := 2.452952;
   DATA[2679,8] := 2.0;
   DATA[2679,9] := 2.0;
   DATA[2679,10] := 2.0;
   DATA[2679,11] := 19.74838;
   DATA[2679,12] := 2.209397;
   DATA[2679,13] := 835.0023;
   DATA[2679,14] := 1.0;
   DATA[2679,15] := 2.0;
   DATA[2679,16] := 1.0;
   DATA[2679,17] := 1.0;
   DATA[2679,18] := 1.0;
   DATA[2679,19] := 2.0;
   DATA[2679,20] := 148.808;
   DATA[2679,21] := 155.473;
   DATA[2679,22] := 1.718515;
   DATA[2679,23] := 882.4661;
   DATA[2679,24] := 2.0;
   DATA[2679,25] := 2.0;
   DATA[2679,26] := 7.874135;
   DATA[2679,27] := 144.7065;
   DATA[2679,28] := 261.3432;
   DATA[2679,29] := 12.07383;
   DATA[2679,30] := 1.731735;
   DATA[2679,31] := 1.307416;
   DATA[2679,32] := 0.7352687;
   DATA[2679,33] := 0.3084905;
   DATA[2679,34] := 2.0;
   DATA[2679,35] := 250.4967;
   DATA[2679,36] := 1.730048;
   DATA[2679,37] := 189.2624;
   DATA[2679,38] := 0.000128152;
   DATA[2679,39] := 1.0;
   DATA[2679,40] := 1.0;
   DATA[2680,0] := 2.552285;
   DATA[2680,1] := 870.7047;
   DATA[2680,3] := 2.0;
   DATA[2680,4] := 262.3366;
   DATA[2680,5] := 8.396757;
   DATA[2680,6] := 329.0182;
   DATA[2680,7] := 2.452568;
   DATA[2680,8] := 2.0;
   DATA[2680,9] := 2.0;
   DATA[2680,10] := 2.0;
   DATA[2680,11] := 19.74838;
   DATA[2680,12] := 2.20645;
   DATA[2680,13] := 834.762;
   DATA[2680,14] := 1.0;
   DATA[2680,15] := 2.0;
   DATA[2680,16] := 1.0;
   DATA[2680,17] := 1.0;
   DATA[2680,18] := 1.0;
   DATA[2680,19] := 2.0;
   DATA[2680,20] := 148.808;
   DATA[2680,21] := 155.4473;
   DATA[2680,22] := 1.718515;
   DATA[2680,23] := 882.5045;
   DATA[2680,24] := 2.0;
   DATA[2680,25] := 2.0;
   DATA[2680,26] := 7.870931;
   DATA[2680,27] := 144.7834;
   DATA[2680,28] := 261.3432;
   DATA[2680,29] := 12.07383;
   DATA[2680,30] := 1.731735;
   DATA[2680,31] := 1.320994;
   DATA[2680,32] := 0.7352687;
   DATA[2680,33] := 0.3084905;
   DATA[2680,34] := 2.0;
   DATA[2680,35] := 250.4967;
   DATA[2680,36] := 1.730048;
   DATA[2680,37] := 189.2624;
   DATA[2680,38] := 0.000128152;
   DATA[2680,39] := 1.0;
   DATA[2680,40] := 1.0;
   DATA[2681,0] := 2.499119;
   DATA[2681,1] := 870.8224;
   DATA[2681,3] := 2.0;
   DATA[2681,4] := 262.3366;
   DATA[2681,5] := 8.396757;
   DATA[2681,6] := 329.0182;
   DATA[2681,7] := 2.451671;
   DATA[2681,8] := 2.0;
   DATA[2681,9] := 2.0;
   DATA[2681,10] := 2.0;
   DATA[2681,11] := 19.74838;
   DATA[2681,12] := 2.20645;
   DATA[2681,13] := 834.6818;
   DATA[2681,14] := 1.0;
   DATA[2681,15] := 2.0;
   DATA[2681,16] := 1.0;
   DATA[2681,17] := 1.0;
   DATA[2681,18] := 1.0;
   DATA[2681,19] := 2.0;
   DATA[2681,20] := 148.808;
   DATA[2681,21] := 155.4473;
   DATA[2681,22] := 1.718515;
   DATA[2681,23] := 882.12;
   DATA[2681,24] := 2.0;
   DATA[2681,25] := 2.0;
   DATA[2681,26] := 7.870931;
   DATA[2681,27] := 144.7834;
   DATA[2681,28] := 261.3432;
   DATA[2681,29] := 12.07383;
   DATA[2681,30] := 1.731735;
   DATA[2681,31] := 1.329064;
   DATA[2681,32] := 0.7352687;
   DATA[2681,33] := 0.3084905;
   DATA[2681,34] := 2.0;
   DATA[2681,35] := 250.4967;
   DATA[2681,36] := 1.730048;
   DATA[2681,37] := 189.2624;
   DATA[2681,38] := 0.000128152;
   DATA[2681,39] := 1.0;
   DATA[2681,40] := 1.0;
   DATA[2682,0] := 2.400154;
   DATA[2682,1] := 870.6654;
   DATA[2682,2] := 1.0;
   DATA[2682,3] := 2.0;
   DATA[2682,4] := 262.3366;
   DATA[2682,5] := 8.396757;
   DATA[2682,6] := 329.0182;
   DATA[2682,7] := 2.451671;
   DATA[2682,8] := 2.0;
   DATA[2682,9] := 2.0;
   DATA[2682,10] := 2.0;
   DATA[2682,11] := 19.74838;
   DATA[2682,12] := 2.20645;
   DATA[2682,13] := 835.2025;
   DATA[2682,14] := 1.0;
   DATA[2682,15] := 2.0;
   DATA[2682,16] := 1.0;
   DATA[2682,17] := 1.0;
   DATA[2682,18] := 1.0;
   DATA[2682,19] := 2.0;
   DATA[2682,20] := 148.808;
   DATA[2682,21] := 155.4473;
   DATA[2682,22] := 1.718515;
   DATA[2682,23] := 882.2738;
   DATA[2682,24] := 2.0;
   DATA[2682,25] := 2.0;
   DATA[2682,26] := 7.873815;
   DATA[2682,27] := 144.7834;
   DATA[2682,28] := 261.3432;
   DATA[2682,29] := 12.07383;
   DATA[2682,30] := 1.731351;
   DATA[2682,31] := 1.332138;
   DATA[2682,32] := 0.7352687;
   DATA[2682,33] := 0.3084905;
   DATA[2682,34] := 2.0;
   DATA[2682,35] := 250.4967;
   DATA[2682,36] := 1.730048;
   DATA[2682,37] := 189.2624;
   DATA[2682,38] := 0.000128152;
   DATA[2682,39] := 1.0;
   DATA[2682,40] := 1.0;
   DATA[2683,0] := 2.223361;
   DATA[2683,1] := 870.9794;
   DATA[2683,2] := 1.0;
   DATA[2683,3] := 2.0;
   DATA[2683,4] := 262.3366;
   DATA[2683,5] := 8.396757;
   DATA[2683,6] := 329.0182;
   DATA[2683,7] := 2.451671;
   DATA[2683,8] := 2.0;
   DATA[2683,9] := 2.0;
   DATA[2683,10] := 2.0;
   DATA[2683,11] := 19.74838;
   DATA[2683,12] := 2.20645;
   DATA[2683,13] := 834.6818;
   DATA[2683,14] := 1.0;
   DATA[2683,15] := 2.0;
   DATA[2683,16] := 1.0;
   DATA[2683,17] := 1.0;
   DATA[2683,18] := 1.0;
   DATA[2683,19] := 2.0;
   DATA[2683,20] := 148.808;
   DATA[2683,21] := 155.4473;
   DATA[2683,22] := 1.718515;
   DATA[2683,23] := 882.5045;
   DATA[2683,24] := 2.0;
   DATA[2683,25] := 2.0;
   DATA[2683,26] := 7.874776;
   DATA[2683,27] := 144.7834;
   DATA[2683,28] := 261.3432;
   DATA[2683,29] := 12.07383;
   DATA[2683,30] := 1.731351;
   DATA[2683,31] := 1.31523;
   DATA[2683,32] := 0.7352687;
   DATA[2683,33] := 0.3084905;
   DATA[2683,34] := 2.0;
   DATA[2683,35] := 250.4967;
   DATA[2683,36] := 1.810143;
   DATA[2683,37] := 189.2624;
   DATA[2683,38] := 0.000128152;
   DATA[2683,39] := 1.0;
   DATA[2683,40] := 1.0;
   DATA[2684,0] := 1.916216;
   DATA[2684,1] := 870.5869;
   DATA[2684,2] := 1.0;
   DATA[2684,3] := 2.0;
   DATA[2684,4] := 262.3366;
   DATA[2684,5] := 8.396757;
   DATA[2684,6] := 329.0182;
   DATA[2684,7] := 2.451671;
   DATA[2684,8] := 2.0;
   DATA[2684,9] := 2.0;
   DATA[2684,10] := 2.0;
   DATA[2684,11] := 19.74838;
   DATA[2684,12] := 2.207091;
   DATA[2684,13] := 835.2025;
   DATA[2684,14] := 1.0;
   DATA[2684,15] := 2.0;
   DATA[2684,16] := 1.0;
   DATA[2684,17] := 1.0;
   DATA[2684,18] := 1.0;
   DATA[2684,19] := 2.0;
   DATA[2684,20] := 148.808;
   DATA[2684,21] := 155.3961;
   DATA[2684,22] := 1.716592;
   DATA[2684,23] := 882.5045;
   DATA[2684,24] := 2.0;
   DATA[2684,25] := 2.0;
   DATA[2684,26] := 7.874776;
   DATA[2684,27] := 144.7834;
   DATA[2684,28] := 261.3432;
   DATA[2684,29] := 12.07383;
   DATA[2684,30] := 1.729557;
   DATA[2684,31] := 1.311387;
   DATA[2684,32] := 0.7352687;
   DATA[2684,33] := 0.3084905;
   DATA[2684,34] := 2.0;
   DATA[2684,35] := 250.4967;
   DATA[2684,36] := 1.810143;
   DATA[2684,37] := 189.2624;
   DATA[2684,38] := 0.000128152;
   DATA[2684,39] := 1.0;
   DATA[2684,40] := 1.0;
   DATA[2685,0] := 1.582808;
   DATA[2685,1] := 870.8224;
   DATA[2685,2] := 1.0;
   DATA[2685,3] := 2.0;
   DATA[2685,4] := 262.3366;
   DATA[2685,5] := 8.396757;
   DATA[2685,6] := 329.0182;
   DATA[2685,7] := 2.452952;
   DATA[2685,8] := 2.0;
   DATA[2685,9] := 2.0;
   DATA[2685,10] := 2.0;
   DATA[2685,11] := 19.74838;
   DATA[2685,12] := 2.208756;
   DATA[2685,13] := 834.842;
   DATA[2685,14] := 1.0;
   DATA[2685,15] := 2.0;
   DATA[2685,16] := 1.0;
   DATA[2685,17] := 1.0;
   DATA[2685,18] := 1.0;
   DATA[2685,19] := 2.0;
   DATA[2685,20] := 148.808;
   DATA[2685,21] := 155.3961;
   DATA[2685,22] := 1.716592;
   DATA[2685,23] := 882.2738;
   DATA[2685,24] := 2.0;
   DATA[2685,25] := 2.0;
   DATA[2685,26] := 7.874776;
   DATA[2685,27] := 144.7834;
   DATA[2685,28] := 261.3432;
   DATA[2685,29] := 12.07383;
   DATA[2685,30] := 1.729557;
   DATA[2685,31] := 1.302677;
   DATA[2685,32] := 0.7352687;
   DATA[2685,33] := 0.3066329;
   DATA[2685,34] := 2.0;
   DATA[2685,35] := 250.4967;
   DATA[2685,36] := 1.810143;
   DATA[2685,37] := 189.2624;
   DATA[2685,38] := 0.000128152;
   DATA[2685,39] := 1.0;
   DATA[2685,40] := 1.0;
   DATA[2686,0] := 1.178618;
   DATA[2686,1] := 870.4299;
   DATA[2686,2] := 1.0;
   DATA[2686,3] := 2.0;
   DATA[2686,4] := 262.3366;
   DATA[2686,5] := 8.396757;
   DATA[2686,6] := 329.0182;
   DATA[2686,7] := 2.452952;
   DATA[2686,8] := 2.0;
   DATA[2686,9] := 2.0;
   DATA[2686,10] := 2.0;
   DATA[2686,11] := 19.69076;
   DATA[2686,12] := 2.209525;
   DATA[2686,13] := 835.1625;
   DATA[2686,14] := 1.0;
   DATA[2686,15] := 2.0;
   DATA[2686,16] := 1.0;
   DATA[2686,17] := 1.0;
   DATA[2686,18] := 1.0;
   DATA[2686,19] := 2.0;
   DATA[2686,20] := 148.808;
   DATA[2686,21] := 155.3961;
   DATA[2686,22] := 1.716592;
   DATA[2686,23] := 882.2738;
   DATA[2686,24] := 2.0;
   DATA[2686,25] := 2.0;
   DATA[2686,26] := 7.874776;
   DATA[2686,27] := 144.7834;
   DATA[2686,28] := 261.3432;
   DATA[2686,29] := 11.84312;
   DATA[2686,30] := 1.729557;
   DATA[2686,31] := 1.292814;
   DATA[2686,32] := 0.7352687;
   DATA[2686,33] := 0.3081703;
   DATA[2686,34] := 2.0;
   DATA[2686,35] := 250.4967;
   DATA[2686,36] := 1.730048;
   DATA[2686,37] := 189.2624;
   DATA[2686,38] := 0.000128152;
   DATA[2686,39] := 1.0;
   DATA[2686,40] := 1.0;
   DATA[2687,0] := 0.801012;
   DATA[2687,1] := 870.1944;
   DATA[2687,2] := 1.0;
   DATA[2687,3] := 2.0;
   DATA[2687,4] := 262.3366;
   DATA[2687,5] := 8.396757;
   DATA[2687,6] := 329.0182;
   DATA[2687,7] := 2.452952;
   DATA[2687,8] := 2.0;
   DATA[2687,9] := 2.0;
   DATA[2687,10] := 2.0;
   DATA[2687,11] := 19.69076;
   DATA[2687,12] := 2.209653;
   DATA[2687,13] := 835.0423;
   DATA[2687,14] := 1.0;
   DATA[2687,15] := 2.0;
   DATA[2687,16] := 1.0;
   DATA[2687,17] := 1.0;
   DATA[2687,18] := 1.0;
   DATA[2687,19] := 2.0;
   DATA[2687,20] := 148.808;
   DATA[2687,21] := 155.3961;
   DATA[2687,22] := 1.716592;
   DATA[2687,23] := 882.5814;
   DATA[2687,24] := 2.0;
   DATA[2687,25] := 2.0;
   DATA[2687,26] := 7.874776;
   DATA[2687,27] := 144.7834;
   DATA[2687,28] := 261.3432;
   DATA[2687,29] := 11.84312;
   DATA[2687,30] := 1.729557;
   DATA[2687,31] := 1.27834;
   DATA[2687,32] := 0.7352687;
   DATA[2687,33] := 0.3086827;
   DATA[2687,34] := 2.0;
   DATA[2687,35] := 250.4967;
   DATA[2687,36] := 1.730048;
   DATA[2687,37] := 189.2624;
   DATA[2687,38] := 0.000128152;
   DATA[2687,39] := 1.0;
   DATA[2687,40] := 1.0;
   DATA[2688,0] := 0.4829773;
   DATA[2688,1] := 869.8411;
   DATA[2688,2] := 1.0;
   DATA[2688,3] := 2.0;
   DATA[2688,4] := 262.3366;
   DATA[2688,5] := 8.396757;
   DATA[2688,6] := 329.0182;
   DATA[2688,7] := 2.452952;
   DATA[2688,8] := 2.0;
   DATA[2688,9] := 2.0;
   DATA[2688,10] := 2.0;
   DATA[2688,11] := 19.69076;
   DATA[2688,12] := 2.209653;
   DATA[2688,13] := 835.0423;
   DATA[2688,14] := 1.0;
   DATA[2688,15] := 2.0;
   DATA[2688,16] := 1.0;
   DATA[2688,17] := 1.0;
   DATA[2688,18] := 1.0;
   DATA[2688,19] := 2.0;
   DATA[2688,20] := 148.808;
   DATA[2688,21] := 155.3961;
   DATA[2688,22] := 1.716464;
   DATA[2688,23] := 882.8505;
   DATA[2688,24] := 2.0;
   DATA[2688,25] := 2.0;
   DATA[2688,26] := 7.874776;
   DATA[2688,27] := 144.7834;
   DATA[2688,28] := 261.3432;
   DATA[2688,29] := 11.84312;
   DATA[2688,30] := 1.729557;
   DATA[2688,31] := 1.257589;
   DATA[2688,32] := 0.7352687;
   DATA[2688,33] := 0.3086827;
   DATA[2688,34] := 2.0;
   DATA[2688,35] := 250.4967;
   DATA[2688,36] := 1.730048;
   DATA[2688,37] := 189.2624;
   DATA[2688,38] := 0.000128152;
   DATA[2688,39] := 1.0;
   DATA[2688,40] := 1.0;
   DATA[2689,0] := 0.2844057;
   DATA[2689,1] := 869.8804;
   DATA[2689,2] := 1.0;
   DATA[2689,3] := 2.0;
   DATA[2689,4] := 262.3366;
   DATA[2689,5] := 8.396757;
   DATA[2689,6] := 329.0182;
   DATA[2689,7] := 2.452952;
   DATA[2689,8] := 2.0;
   DATA[2689,9] := 2.0;
   DATA[2689,10] := 2.0;
   DATA[2689,11] := 19.69076;
   DATA[2689,12] := 2.209653;
   DATA[2689,13] := 835.2426;
   DATA[2689,14] := 1.0;
   DATA[2689,15] := 2.0;
   DATA[2689,16] := 1.0;
   DATA[2689,17] := 1.0;
   DATA[2689,18] := 1.0;
   DATA[2689,19] := 2.0;
   DATA[2689,20] := 148.808;
   DATA[2689,21] := 155.3961;
   DATA[2689,22] := 1.716464;
   DATA[2689,23] := 882.7736;
   DATA[2689,24] := 2.0;
   DATA[2689,25] := 2.0;
   DATA[2689,26] := 7.874776;
   DATA[2689,27] := 144.7834;
   DATA[2689,28] := 261.3432;
   DATA[2689,29] := 12.07383;
   DATA[2689,30] := 1.729557;
   DATA[2689,31] := 1.245805;
   DATA[2689,32] := 0.7352687;
   DATA[2689,33] := 0.3086827;
   DATA[2689,34] := 2.0;
   DATA[2689,35] := 250.3525;
   DATA[2689,36] := 1.730048;
   DATA[2689,37] := 189.1342;
   DATA[2689,38] := 0.000128152;
   DATA[2689,39] := 1.0;
   DATA[2689,40] := 1.0;
   DATA[2690,0] := 0.1518112;
   DATA[2690,1] := 869.8019;
   DATA[2690,2] := 1.0;
   DATA[2690,3] := 2.0;
   DATA[2690,4] := 262.3366;
   DATA[2690,5] := 8.396757;
   DATA[2690,6] := 329.0182;
   DATA[2690,7] := 2.452952;
   DATA[2690,8] := 2.0;
   DATA[2690,9] := 2.0;
   DATA[2690,10] := 2.0;
   DATA[2690,11] := 19.70677;
   DATA[2690,12] := 2.209653;
   DATA[2690,13] := 835.2025;
   DATA[2690,14] := 1.0;
   DATA[2690,15] := 2.0;
   DATA[2690,16] := 1.0;
   DATA[2690,17] := 1.0;
   DATA[2690,18] := 1.0;
   DATA[2690,19] := 2.0;
   DATA[2690,20] := 148.808;
   DATA[2690,21] := 155.3961;
   DATA[2690,22] := 1.716464;
   DATA[2690,23] := 882.7736;
   DATA[2690,24] := 2.0;
   DATA[2690,25] := 2.0;
   DATA[2690,26] := 7.874776;
   DATA[2690,27] := 144.7834;
   DATA[2690,28] := 261.3432;
   DATA[2690,29] := 12.22763;
   DATA[2690,30] := 1.731479;
   DATA[2690,31] := 1.244652;
   DATA[2690,32] := 0.7352687;
   DATA[2690,33] := 0.3086827;
   DATA[2690,34] := 2.0;
   DATA[2690,35] := 250.3525;
   DATA[2690,36] := 1.730048;
   DATA[2690,37] := 189.1342;
   DATA[2690,38] := 0.000128152;
   DATA[2690,39] := 1.0;
   DATA[2690,40] := 1.0;
   DATA[2691,0] := 0.07334337;
   DATA[2691,1] := 869.8411;
   DATA[2691,2] := 1.0;
   DATA[2691,3] := 2.0;
   DATA[2691,4] := 262.3366;
   DATA[2691,5] := 8.396757;
   DATA[2691,6] := 329.1207;
   DATA[2691,7] := 2.452952;
   DATA[2691,8] := 2.0;
   DATA[2691,9] := 2.0;
   DATA[2691,10] := 2.0;
   DATA[2691,11] := 19.74198;
   DATA[2691,12] := 2.209653;
   DATA[2691,13] := 835.4429;
   DATA[2691,14] := 1.0;
   DATA[2691,15] := 2.0;
   DATA[2691,16] := 1.0;
   DATA[2691,17] := 1.0;
   DATA[2691,18] := 1.0;
   DATA[2691,19] := 2.0;
   DATA[2691,20] := 148.808;
   DATA[2691,21] := 155.3961;
   DATA[2691,22] := 1.718515;
   DATA[2691,23] := 882.5045;
   DATA[2691,24] := 2.0;
   DATA[2691,25] := 2.0;
   DATA[2691,26] := 7.874776;
   DATA[2691,27] := 144.7834;
   DATA[2691,28] := 261.3432;
   DATA[2691,29] := 12.22763;
   DATA[2691,30] := 1.731479;
   DATA[2691,31] := 1.262713;
   DATA[2691,32] := 0.7352687;
   DATA[2691,33] := 0.3074016;
   DATA[2691,34] := 2.0;
   DATA[2691,35] := 250.2724;
   DATA[2691,36] := 1.730048;
   DATA[2691,37] := 188.958;
   DATA[2691,38] := 0.000128152;
   DATA[2691,39] := 1.0;
   DATA[2691,40] := 1.0;
   DATA[2692,0] := 0.02370048;
   DATA[2692,1] := 869.7234;
   DATA[2692,2] := 1.0;
   DATA[2692,3] := 2.0;
   DATA[2692,4] := 262.3366;
   DATA[2692,5] := 8.396757;
   DATA[2692,6] := 329.1207;
   DATA[2692,7] := 2.452952;
   DATA[2692,8] := 2.0;
   DATA[2692,9] := 2.0;
   DATA[2692,10] := 2.0;
   DATA[2692,11] := 19.74198;
   DATA[2692,12] := 2.209653;
   DATA[2692,13] := 835.4028;
   DATA[2692,14] := 1.0;
   DATA[2692,15] := 2.0;
   DATA[2692,16] := 1.0;
   DATA[2692,17] := 1.0;
   DATA[2692,18] := 1.0;
   DATA[2692,19] := 2.0;
   DATA[2692,20] := 148.808;
   DATA[2692,21] := 155.3961;
   DATA[2692,22] := 1.718515;
   DATA[2692,23] := 882.2738;
   DATA[2692,24] := 2.0;
   DATA[2692,25] := 2.0;
   DATA[2692,26] := 7.874776;
   DATA[2692,27] := 144.7834;
   DATA[2692,28] := 261.3432;
   DATA[2692,29] := 12.22763;
   DATA[2692,30] := 1.729172;
   DATA[2692,31] := 1.271423;
   DATA[2692,32] := 0.7352687;
   DATA[2692,33] := 0.3075937;
   DATA[2692,34] := 2.0;
   DATA[2692,35] := 250.2724;
   DATA[2692,36] := 1.730048;
   DATA[2692,37] := 188.958;
   DATA[2692,38] := 0.000128152;
   DATA[2692,39] := 1.0;
   DATA[2692,40] := 1.0;
   DATA[2693,0] := 0.000640553;
   DATA[2693,1] := 869.7234;
   DATA[2693,2] := 1.0;
   DATA[2693,3] := 2.0;
   DATA[2693,4] := 262.3366;
   DATA[2693,5] := 8.396757;
   DATA[2693,6] := 329.1464;
   DATA[2693,7] := 2.452952;
   DATA[2693,8] := 2.0;
   DATA[2693,9] := 2.0;
   DATA[2693,10] := 2.0;
   DATA[2693,11] := 19.74198;
   DATA[2693,12] := 2.207091;
   DATA[2693,13] := 835.8033;
   DATA[2693,14] := 1.0;
   DATA[2693,15] := 2.0;
   DATA[2693,16] := 1.0;
   DATA[2693,17] := 1.0;
   DATA[2693,18] := 1.0;
   DATA[2693,19] := 2.0;
   DATA[2693,20] := 148.808;
   DATA[2693,21] := 155.3961;
   DATA[2693,22] := 1.718515;
   DATA[2693,23] := 882.8121;
   DATA[2693,24] := 2.0;
   DATA[2693,25] := 2.0;
   DATA[2693,26] := 7.874776;
   DATA[2693,27] := 144.7834;
   DATA[2693,28] := 261.3432;
   DATA[2693,29] := 12.22763;
   DATA[2693,30] := 1.729172;
   DATA[2693,31] := 1.272064;
   DATA[2693,32] := 0.7352687;
   DATA[2693,33] := 0.3082983;
   DATA[2693,34] := 2.0;
   DATA[2693,35] := 250.2724;
   DATA[2693,36] := 1.730048;
   DATA[2693,37] := 188.958;
   DATA[2693,38] := 0.000128152;
   DATA[2693,39] := 1.0;
   DATA[2693,40] := 1.0;
END_DATA_BLOCK

DATA_BLOCK "DB_Main"   // DB6
{ S7_Optimized_Access := 'TRUE' }
VERSION : 0.1
   VAR
      iState : Int;
      PredictCount : Int;
      bStart : Bool;
      Mse : Real;
   END_VAR
BEGIN
END_DATA_BLOCK

DATA_BLOCK "DB_FeatureNormRef_Means"   // DB7
{ S7_Optimized_Access := 'TRUE' }
VERSION : 0.1
   VAR
      Means : Array[0..39] of Real;
   END_VAR
BEGIN
   Means[0] := 1.846544;
   Means[1] := 582.3317;
   Means[2] := 1.719179;
   Means[3] := 1.744085;
   Means[4] := 262.3805;
   Means[5] := 8.393863;
   Means[6] := 361.9682;
   Means[7] := 1.824498;
   Means[8] := 1.741861;
   Means[9] := 1.742247;
   Means[10] := 1.599953;
   Means[11] := 16.52142;
   Means[12] := 1.820565;
   Means[13] := 891.7278;
   Means[14] := 1.005415;
   Means[15] := 1.795682;
   Means[16] := 1.019948;
   Means[17] := 1.024403;
   Means[18] := 1.006612;
   Means[19] := 1.813745;
   Means[20] := 107.9063;
   Means[21] := 178.6221;
   Means[22] := 1.683628;
   Means[23] := 872.4719;
   Means[24] := 1.989312;
   Means[25] := 1.989295;
   Means[26] := 7.859592;
   Means[27] := 167.5583;
   Means[28] := 265.8126;
   Means[29] := 12.47605;
   Means[30] := 1.693144;
   Means[31] := 1.252732;
   Means[32] := 0.7332894;
   Means[33] := 0.3058438;
   Means[34] := 1.988802;
   Means[35] := 251.657;
   Means[36] := 1.217715;
   Means[37] := 191.1807;
   Means[38] := 0.0142492;
   Means[39] := 1.007837;
END_DATA_BLOCK

DATA_BLOCK "DB_FeatureNormRef_std"   // DB8
{ S7_Optimized_Access := 'TRUE' }
VERSION : 0.1
   VAR
      std : Array[0..39] of Real;
   END_VAR
BEGIN
   std[0] := 1.134874;
   std[1] := 131.2155;
   std[2] := 0.4579044;
   std[3] := 0.436374;
   std[4] := 5.261742;
   std[5] := 0.1128395;
   std[6] := 59.83524;
   std[7] := 1.067913;
   std[8] := 0.4456327;
   std[9] := 0.4373973;
   std[10] := 0.4899075;
   std[11] := 6.801564;
   std[12] := 0.8329131;
   std[13] := 117.8872;
   std[14] := 0.1100685;
   std[15] := 0.419305;
   std[16] := 0.1684625;
   std[17] := 0.1948795;
   std[18] := 0.08104688;
   std[19] := 0.3893126;
   std[20] := 66.43026;
   std[21] := 11.66761;
   std[22] := 0.1758617;
   std[23] := 113.9631;
   std[24] := 0.1028308;
   std[25] := 0.1029105;
   std[26] := 0.06156169;
   std[27] := 11.32486;
   std[28] := 5.737159;
   std[29] := 11.95808;
   std[30] := 0.1767241;
   std[31] := 0.1317653;
   std[32] := 0.0767542;
   std[33] := 0.03271202;
   std[34] := 0.105228;
   std[35] := 25.34136;
   std[36] := 0.2577594;
   std[37] := 19.61726;
   std[38] := 0.1478796;
   std[39] := 0.08817827;
END_DATA_BLOCK

DATA_BLOCK "DB_LSTM_SWAT_BASE"   // DB9
{ S7_Optimized_Access := 'TRUE' }
VERSION : 0.1
// stored: InstanceOfName LSTM_SWAT_BASE
"LSTM_SWAT_BASE"
BEGIN
END_DATA_BLOCK

DATA_BLOCK "DB_Measuring"   // DB10
{ S7_Optimized_Access := 'TRUE' }
VERSION : 0.1
   VAR
      CycleTime_ms : DInt;
      last_cycle_time : LTime;
      last_cycle_ms : Array[0..3000] of DInt;
   END_VAR
BEGIN
END_DATA_BLOCK

// folder: (top level)

FUNCTION "_RestartTesting" : Int   // FC1, SCL
{ S7_Optimized_Access := 'TRUE' }
VERSION : 0.1
   VAR_INPUT
      bStart : Bool;
   END_VAR
BEGIN
   IF #bStart THEN
       "DB_Main".PredictCount := 0;
       "DB_Result".TruePositive := 0;
       "DB_Result".TrueNegative := 0;
       "DB_Result".FalsePositive := 0;
       "DB_Result".FalseNegative := 0;
       #_RestartTesting := 10;
   ELSE
       #_RestartTesting := 0;
   END_IF;
END_FUNCTION

FUNCTION "_Zscore" : Real   // FC7, SCL
{ S7_Optimized_Access := 'TRUE' }
VERSION : 0.1
   VAR_INPUT
      iRow : Int;
      iCol : Int;
   END_VAR
BEGIN
   #_Zscore := ("DB_Attack_v0_first_attack".DATA[#iRow, #iCol] - "DB_FeatureNormRef_Means".Means[#iCol]) / "DB_FeatureNormRef_std".std[#iCol];
END_FUNCTION

ORGANIZATION_BLOCK "Main"   // OB1, SCL, ProgramCycle
TITLE = "Main Program Sweep (Cycle)"
{ S7_Optimized_Access := 'TRUE' }
VERSION : 0.1
   VAR_INPUT
      Initial_Call : Bool;   // Initial call of this OB
      Remanence : Bool;   // =True, if remanent data are available
   END_VAR
   VAR_TEMP
      I : Int;
      j : Int;
      LSTM : Int;
      vInfo : Variant;
      lastCycleTime : DInt;
      retVal : Int;
   END_VAR
BEGIN
           //-->> Cycle Time measuring
   #retVal:= RT_INFO(
                     MODE := 25,
                     OB := 1,
                     INFO := "DB_Measuring".last_cycle_time
   );
   "DB_Measuring".last_cycle_ms["DB_Main".PredictCount]:= LTIME_TO_DINT("DB_Measuring".last_cycle_time);
   "DB_Measuring".CycleTime_ms := LTIME_TO_DINT("DB_Measuring".last_cycle_time) /1000000;



    CASE "DB_Main".iState OF
           //-->> IDLE
       0:
           "DB_Main".iState := "_RestartTesting"("DB_Main".bStart);


           //-->> Fill Model Window
       10:
           FOR #I := 0 TO 99 DO
               FOR #j := 0 TO 39 DO
                   "DB_LSTM_SWAT_BASE".x_t[#I, #j] := "_Zscore"(iRow := #I, iCol := #j);   
               END_FOR;
           END_FOR;
           "DB_Result".TrueNegative := 100;
           "DB_Main".PredictCount := 100;
           "DB_Main".iState := 20;


           //-->> Call LSTM modell
       20:
           "DB_LSTM_SWAT_BASE"(bStart := TRUE,
                               Threshold := "DB_Result".THRESHOLD,
                               predicted_class => "DB_Result".Predicted_class);
           "DB_Main".iState := 30;


           //-->> Predict Ready
       30:
           IF "DB_Result".Predicted_class = 1 AND
               REAL_TO_INT("DB_Attack_v0_first_attack".DATA["DB_Main".PredictCount, 40]) = 1
           THEN
               "DB_Result".TruePositive := "DB_Result".TruePositive + 1;
           ELSIF "DB_Result".Predicted_class = 0 AND
               REAL_TO_INT("DB_Attack_v0_first_attack".DATA["DB_Main".PredictCount, 40]) = 0
           THEN
               "DB_Result".TrueNegative := "DB_Result".TrueNegative + 1;
           ELSIF "DB_Result".Predicted_class = 1 AND
               REAL_TO_INT("DB_Attack_v0_first_attack".DATA["DB_Main".PredictCount, 40]) = 0
           THEN
               "DB_Result".FalsePositive := "DB_Result".FalsePositive + 1;
           ELSIF "DB_Result".Predicted_class = 0 AND
               REAL_TO_INT("DB_Attack_v0_first_attack".DATA["DB_Main".PredictCount, 40]) = 1
           THEN
               "DB_Result".FalseNegative := "DB_Result".FalseNegative + 1;
           END_IF;
           "DB_Main".PredictCount := "DB_Main".PredictCount + 1;

           IF "DB_Main".PredictCount >= "DB_Result".EXPECTED_PREDICITON_COUNT THEN
               "DB_Main".iState  := 100;
           ELSE
               "DB_Main".iState := 40;
           END_IF;


           //-->> ShiftInputWindow
       40:
           FOR #I := 0 TO 15 DO
               "DB_LSTM_SWAT_BASE".h_tm1[#I] := 0.0;
               "DB_LSTM_SWAT_BASE".c_tm1[#I] := 0.0;
           END_FOR;

           FOR #I := 0 TO 98 DO
               FOR #j := 0 TO 39 DO
                   "DB_LSTM_SWAT_BASE".x_t[#I, #j] :="DB_LSTM_SWAT_BASE".x_t[#I + 1, #j];
               END_FOR;
           END_FOR;

           FOR #j := 0 TO 39 DO
               "DB_LSTM_SWAT_BASE".x_t[99, #j] := "_Zscore"(iRow := "DB_Main".PredictCount , iCol := #j);
           END_FOR;
           "DB_Main".iState := 20;


           //-->> Test Ready Compare Result
       100:
           IF "DB_Result".TrueNegative <> "DB_Result".EXPECTED_TRUE_NEGATIVE THEN
               "DB_Result".MismatchCount := "DB_Result".MismatchCount + 1;
           END_IF;
           IF "DB_Result".FalsePositive <>"DB_Result".EXPECTED_FALSE_POSITIVE THEN
               "DB_Result".MismatchCount := "DB_Result".MismatchCount + 1;
           END_IF;
           IF "DB_Result".FalseNegative <> "DB_Result".EXPECTED_FALSE_NEGATIVE THEN
               "DB_Result".MismatchCount := "DB_Result".MismatchCount + 1;
           END_IF;
           IF "DB_Result".TruePositive <> "DB_Result".EXPECTED_TRUE_POSITIVE THEN
               "DB_Result".MismatchCount := "DB_Result".MismatchCount + 1;
           END_IF;
           IF "DB_Main".PredictCount <> "DB_Result".EXPECTED_PREDICITON_COUNT THEN
               "DB_Result".MismatchCount := "DB_Result".MismatchCount + 1;
           END_IF;
           IF "DB_Result".MismatchCount <> 0 THEN
               "DB_Main".iState := 150; 
           ELSE
               "DB_Main".iState := 200; 
           END_IF;

           //-->> Finish   
       150,200:
           IF NOT "DB_Main".bStart THEN
               "DB_Main".iState := 0;
           END_IF;

     END_CASE;
END_ORGANIZATION_BLOCK

// folder: LSTM_SWAT_BASE

FUNCTION_BLOCK "LSTM_SWAT_BASE"   // FB1, SCL
{ S7_Optimized_Access := 'TRUE' }
VERSION : 0.1
   VAR_INPUT
      bStart : Bool;
      x_t : Array[0..99, 0..39] of Real;
      c_tm1 : Array[0..15] of Real;
      h_tm1 : Array[0..15] of Real;
      Threshold : Real;
   END_VAR
   VAR_OUTPUT
      c_t : Array[0..15] of Real;
      h_t : Array[0..15] of Real;
      y : Array[0..39] of Real;
      predicted_class : Int;
   END_VAR
   VAR
      attack : Int := 0;
      normal : Int := 0;
      f_t : Array[0..15] of Real;
      i_t : Array[0..15] of Real;
      g_t : Array[0..15] of Real;
      o_t : Array[0..15] of Real;
      x_i : Real := 0.0;
      x_f : Real := 0.0;
      x_g : Real := 0.0;
      x_o : Real := 0.0;
      x_ct : Real := 0.0;
      i : Int := 0;
      j : Int := 0;
      t : Int := 0;
      max_value : Real := 0.0;
      k : Int := 0;
      msearray : Array[0..3000] of Real;
      err : Real := 0.0;
   END_VAR
BEGIN
   IF #bStart THEN
       FOR #t := 0 TO 99 DO 
           FOR #i := 0 TO 15 DO 
               // Input gate activation 
               #x_i := "DB_model_HS16_IW100".B_i[#i];
               FOR #k := 0 TO 39 DO
                   #x_i := #x_i + "DB_model_HS16_IW100".W_i[#i, #k] * #x_t[#t, #k];
               END_FOR;
               FOR #j := 0 TO 15 DO
                   #x_i := #x_i + "DB_model_HS16_IW100".R_i[#i, #j] * #h_tm1[#j];
               END_FOR;
               #x_i := "_LIMIT"(inVal := #x_i, maxVal := 20, minVal := -20);
               #i_t[#i] := 1.0 / (1.0 + EXP(- #x_i));

               // Forget gate activation 
               #x_f := "DB_model_HS16_IW100".B_f[#i];
               FOR #k := 0 TO 39 DO
                   #x_f := #x_f + "DB_model_HS16_IW100".W_f[#i, #k] * #x_t[#t, #k];
               END_FOR;
               FOR #j := 0 TO 15 DO
                   #x_f := #x_f + "DB_model_HS16_IW100".R_f[#i, #j] * #h_tm1[#j];
               END_FOR;
               #x_f := "_LIMIT"(inVal := #x_f, maxVal := 20, minVal := -20);
               #f_t[#i] := 1.0 / (1.0 + EXP(- #x_f));

               // Cell candidate activation (tanh)
               #x_g := "DB_model_HS16_IW100".B_g[#i];
               FOR #k := 0 TO 39 DO
                   #x_g := #x_g + "DB_model_HS16_IW100".W_g[#i, #k] * #x_t[#t, #k];
               END_FOR;
               FOR #j := 0 TO 15 DO
                   #x_g := #x_g + "DB_model_HS16_IW100".R_g[#i, #j] * #h_tm1[#j];
               END_FOR;
               #x_g := "_LIMIT"(inVal := #x_g, maxVal := 20, minVal := -20);
               #g_t[#i] := (EXP(#x_g) - EXP(- #x_g)) / (EXP(#x_g) + EXP(- #x_g));


               // Output gate activation (sigmoid)
               #x_o := "DB_model_HS16_IW100".B_o[#i];
               FOR #k := 0 TO 39 DO
                   #x_o := #x_o + "DB_model_HS16_IW100".W_o[#i, #k] * #x_t[#t, #k];
               END_FOR;
               FOR #j := 0 TO 15 DO
                   #x_o := #x_o + "DB_model_HS16_IW100".R_o[#i, #j] * #h_tm1[#j];
               END_FOR;
               #x_o := "_LIMIT"(inVal := #x_o, maxVal := 20, minVal := -20);
               #o_t[#i] := 1.0 / (1.0 + EXP(- #x_o));

               // Update cell state
               #c_t[#i] := #f_t[#i] * #c_tm1[#i] + #i_t[#i] * #g_t[#i];

               // Update hidden state (tanh)
               #x_ct := "_LIMIT"(inVal := #c_t[#i], maxVal := 20, minVal := -20);
               #h_t[#i] := #o_t[#i] * ((EXP(#x_ct) - EXP(- #x_ct)) / (EXP(#x_ct) + EXP(- #x_ct)));
           END_FOR;

           FOR #i := 0 TO 15 DO // Shift LSTM states to next time step
               #c_tm1[#i] := #c_t[#i];
               #h_tm1[#i] := #h_t[#i];
           END_FOR;
       END_FOR;

       // Fully connected layer for reconstruction (not classification)
       "_FC_layer"(h_t := #h_t,
                   y => #y); 

       // Reconstruction error (MSE) calculation
       "DB_Main".Mse := 0.0;
       FOR #k := 0 TO 39 DO
           "DB_Main".Mse := "DB_Main".Mse + (#x_t[99, #k] - #y[#k]) * (#x_t[99, #k] - #y[#k]);
       END_FOR;

       // Attack/Normal detection
       "DB_Main".Mse := "DB_Main".Mse / INT_TO_REAL(40);
       IF "DB_Main".Mse > #Threshold THEN
           #predicted_class := 1; // Attack
       ELSE
           #predicted_class := 0; // Normal
       END_IF;
   END_IF;
END_FUNCTION_BLOCK

FUNCTION "_FC_layer" : Void   // FC2, SCL
{ S7_Optimized_Access := 'TRUE' }
VERSION : 0.1
   VAR_INPUT
      h_t : Array[0..15] of Real;
   END_VAR
   VAR_OUTPUT
      y : Array[0..39] of Real;
   END_VAR
   VAR_TEMP
      i : Int;
      j : Int;
   END_VAR
BEGIN
   FOR #i := 0 TO 39 DO
       #y[#i] := 0.0;
       FOR #j := 0 TO 15 DO
           #y[#i] := #y[#i] + "DB_model_HS16_IW100".FC_W[#i, #j] * #h_t[#j];
       END_FOR;
       #y[#i] := #y[#i] + "DB_model_HS16_IW100".FC_B[#i];
   END_FOR;
END_FUNCTION

FUNCTION "_Sigmoid" : Real   // FC3, SCL
{ S7_Optimized_Access := 'TRUE' }
VERSION : 0.1
   VAR_INPUT
      x : Real;
   END_VAR
   VAR_TEMP
      "e" : Real;
   END_VAR
BEGIN
   IF #x >= 0.0 THEN
       #_Sigmoid := 1.0 / (1.0 + EXP(- #x));
   ELSE
       #e := EXP(#x);
       #_Sigmoid := #e / (1.0 + #e);
   END_IF;
END_FUNCTION

FUNCTION "_TANH" : Real   // FC4, SCL
{ S7_Optimized_Access := 'TRUE' }
VERSION : 0.1
   VAR_INPUT
      x : Real;
   END_VAR
   VAR_TEMP
      "e" : Real;
   END_VAR
BEGIN
   IF #x > 10.0 THEN
       #_TANH := 1.0;
   ELSIF #x < -10.0 THEN
       #_TANH := -1.0;
   ELSE
       #e := EXP(-2.0 * #x);
       #_TANH := (1.0 - #e) / (1.0 + #e);
   END_IF;
END_FUNCTION

FUNCTION "_LIMIT" : Real   // FC5, SCL
{ S7_Optimized_Access := 'TRUE' }
VERSION : 0.1
   VAR_INPUT
      inVal : Real;
      minVal : Real;
      maxVal : Real;
   END_VAR
   VAR_TEMP
      lo : Real;
      hi : Real;
   END_VAR
BEGIN
   IF #inVal < #minVal THEN
       #_LIMIT := #minVal;
   ELSIF #inVal > #maxVal THEN
       #_LIMIT := #maxVal;
   ELSE
       #_LIMIT := #inVal;
   END_IF;
END_FUNCTION